// TwinCAT 3 PLC project JOGAN
// ProgramVersion: 3.1.4020.4
// libraries:
//   Tc2_Standard, * (Beckhoff Automation GmbH)
//   Tc2_System, * (Beckhoff Automation GmbH)
//   Tc3_Module, * (Beckhoff Automation GmbH)
// project tree:
//   DUTs/ T_MACHINE_POSITION.TcDUT, T_CURRENT_TRANSACTION.TcDUT, T_JIG_SOCKET.TcDUT
//   GVLs/ FLAG_VAR.TcGVL, INDEXING_1_VAR.TcGVL, INDEXING_2_VAR.TcGVL, INPUT_G6_VAR.TcGVL, INPUT_VAR.TcGVL, LOADER_RS4_VAR.TcGVL, LOADER_VAR.TcGVL, POWER_CONTROL.TcGVL, SORTER_RS4_VAR.TcGVL, SORTER_VAR.TcGVL, TESTER_C8_VAR.TcGVL
//   / PlcTask.TcTTO (not stored)
//   POUs/ EXECUTE_FUNCTION.TcPOU (not stored), MAIN.TcPOU, STQWE.TcPOU
//   POUs/FUKUDA/ FUKUDA_MOVE.TcPOU, FUKUDA_MOVE_1.TcPOU, INPUT_PROG.TcPOU, LOAD_FUKUDA.TcPOU, LOAD_FUKUDA_1.TcPOU, RETURN_FUKUDA.TcPOU, RETURN_FUKUDA_1.TcPOU (not stored)
//   POUs/LASER/ LASER_MOVE.TcPOU, LASER_PROG.TcPOU, LOAD_LASER.TcPOU, LOAD_NG.TcPOU, RETURN_LASER.TcPOU, RETURN_NG.TcPOU
//   POUs/LOADER/ INDEXING.TcPOU, INDEX_1.TcPOU, INDEXING_2.TcPOU, STRAIGHTENING_PROG_1.TcPOU, STR.TcPOU (not stored)
//   POUs/ROBOT/ INPUT_G6.TcPOU, TESTER_C8.TcPOU, LOADER_RS4.TcPOU, SORTER_RS4.TcPOU
// real-time tasks:
//   TASK PlcTask: cycle T#10ms, priority 20, ADS port 350
// I/O:
//   DEVICE Device 5 (EtherCAT), AmsNetId 172.18.128.227.6.1
//     Term 1 (EK1100) [EK1100 EtherCAT Coupler (2A E-Bus)]
//       Term 2 (EL1808) [EL1808 8Ch. Dig. Input 24V, 3ms]
//       Term 3 (EL1808) [EL1808 8Ch. Dig. Input 24V, 3ms]
//       Term 4 (EL1808) [EL1808 8Ch. Dig. Input 24V, 3ms]
//       Term 5 (EL1808) [EL1808 8Ch. Dig. Input 24V, 3ms]
//       Term 6 (EL2808) [EL2808 8Ch. Dig. Output 24V, 0.5A]
//       Term 7 (EL2808) [EL2808 8Ch. Dig. Output 24V, 0.5A]
//       Term 8 (EL2808) [EL2808 8Ch. Dig. Output 24V, 0.5A]
//       Term 9 (EL2808) [EL2808 8Ch. Dig. Output 24V, 0.5A]
//       Term 10 (EL2808) [EL2808 8Ch. Dig. Output 24V, 0.5A]
//       Term 11 (EL3058) [EL3058 8Ch. Ana. Input 4-20mA]
//       Term 12 (EL1904) [EL1904, 4 Ch. Safety Input 24V, TwinSAFE]
//         modules: Module 1 (FSOES)
//       Term 13 (EL1904) [EL1904, 4 Ch. Safety Input 24V, TwinSAFE]
//         modules: Module 1 (FSOES)
//       Term 14 (EL6731) [EL6731 PROFIBUS DP Master]
//       Term 15 (EK1110) [EK1110 EtherCAT extension]
//     Term 16 (EK1100) [EK1100 EtherCAT Coupler (2A E-Bus)]
//       Term 17 (EL1808) [EL1808 8Ch. Dig. Input 24V, 3ms]
//       Term 18 (EL1808) [EL1808 8Ch. Dig. Input 24V, 3ms]
//       Term 19 (EL1808) [EL1808 8Ch. Dig. Input 24V, 3ms]
//       Term 20 (EL1808) [EL1808 8Ch. Dig. Input 24V, 3ms]
//       Term 21 (EL1808) [EL1808 8Ch. Dig. Input 24V, 3ms]
//       Term 22 (EL1808) [EL1808 8K. Dig. Eingang 24V, 3ms]
//       Term 23 (EL2808) [EL2808 8Ch. Dig. Output 24V, 0.5A]
//       Term 24 (EL2808) [EL2808 8Ch. Dig. Output 24V, 0.5A]
//       Term 25 (EL2808) [EL2808 8Ch. Dig. Output 24V, 0.5A]
//       Term 26 (EL2808) [EL2808 8Ch. Dig. Output 24V, 0.5A]
//       Term 27 (EL2808) [EL2808 8Ch. Dig. Output 24V, 0.5A]
//       Term 28 (EL2808) [EL2808 8Ch. Dig. Output 24V, 0.5A]
//       Term 29 (EL2808) [EL2808 8Ch. Dig. Output 24V, 0.5A]
//       Term 30 (EL2808) [EL2808 8Ch. Dig. Output 24V, 0.5A]
//       Term 31 (EL6731) [EL6731 PROFIBUS DP Master]
//       Term 32 (EK1110) [EK1110 EtherCAT extension]
//     Box 33 (EP2809-0021)RS4-2 [EP2809-0021 16 Ch. Dig. Output 24V, 0,5A, M8]
//     Box 34 (EP1809-0021)RS4-2 [EP1809-0021 16 Ch. Dig. Input 24V, 3ms, M8]
//     Box 35 (EP2809-0021)RS4-1 [EP2809-0021 16 Ch. Dig. Output 24V, 0,5A, M8]
//     Box 36 (EP2809-0021)RS4-1 [EP1809-0021 16 Ch. Dig. Input 24V, 3ms, M8]
//     Box 37 (EP1809-0021)G6 [EP1809-0021 16 Ch. Dig. Input 24V, 3ms, M8]
//     Box 38 (EP2809-0021) G6 [EP2809-0021 16 Ch. Dig. Output 24V, 0,5A, M8]
//     Box 39 (EPSON RC700 EtherCAT Slave)G6 [EPSON RC700 EtherCAT Slave]
//     Box 40 (EPSON RC700 EtherCAT Slave)RS4-1 [EPSON RC700 EtherCAT Slave]
//     Box 40 (EPSON RC700 EtherCAT Slave)C8 [EPSON RC700 EtherCAT Slave]
//     Box 42 (EPSON RC700 EtherCAT Slave)RS4-2 [EPSON RC700 EtherCAT Slave]
//     Box 47 (EP2339-0021) [EP2339-0021 16 Ch. Dig. Input/Output 24V, 0,5A, M8]
//     Box 88 (EP2339-0021) [EP2339-0021 16 Ch. Dig. Input/Output 24V, 0,5A, M8]
//   DEVICE Device 1 (EL6731), AmsNetId 172.18.128.227.2.1
//     Box 43 (LEC-GPR1) // Vendor: SMC Corporation Revision: V1.0
//     Box 44 (AX9000T) INDEXING 1 // Vendor: CKD Corporation Revision: Version 1.000
//      // Vendor: CKD Corporation Revision: Version 1.000
//   DEVICE Device 2 (EL6731), AmsNetId 172.18.128.227.3.1
//     Box 46 (LEC-GPR1) // Vendor: SMC Corporation Revision: V1.0
// variable links:
//   JOGAN/JOGAN Instance <-> Device 1 (EL6731)/
//     PlcTask Inputs/INDEXING_2_VAR.DataByteInput2 <-> Module 1 (8 Bytes Out,8 Bytes In)/Inputs/8 Bytes Out,8 Bytes In_0_0
//     PlcTask Outputs/INDEXING_2_VAR.DataByteOutput2 <-> Module 1 (8 Bytes Out,8 Bytes In)/Outputs/8 Bytes Out,8 Bytes In_1_0
//   JOGAN/JOGAN Instance <-> Device 1 (EL6731)/Box 43 (LEC-GPR1)
//     PlcTask Inputs/INPUT_VAR.DataWordInput1 <-> Module 1 (Input 16 words)/Inputs/Input 16 words_0_0
//     PlcTask Inputs/INPUT_VAR.DataWordInput2 <-> Module 2 (Input 16 words)/Inputs/Input 16 words_0_0
//     PlcTask Inputs/INPUT_VAR.DataWordInput3 <-> Module 3 (Input 16 words)/Inputs/Input 16 words_0_0
//     PlcTask Outputs/INPUT_VAR.DataWordOutput1 <-> Module 5 (Output 16 words)/Outputs/Output 16 words_1_0
//     PlcTask Outputs/INPUT_VAR.DataWordOutput2 <-> Module 6 (Output 16 words)/Outputs/Output 16 words_1_0
//     PlcTask Outputs/INPUT_VAR.DataWordOutput3 <-> Module 7 (Output 16 words)/Outputs/Output 16 words_1_0
//     PlcTask Outputs/INPUT_VAR.DataWordOutput4 <-> Module 8 (Output 9 words)/Outputs/Output 9 words_1_0
//   JOGAN/JOGAN Instance <-> Device 1 (EL6731)/Box 44 (AX9000T) INDEXING 1
//     PlcTask Inputs/INDEXING_1_VAR.DataByteInput <-> Module 2 (8 Bytes Out,8 Bytes In)/Inputs/8 Bytes Out,8 Bytes In_0_0
//     PlcTask Outputs/INDEXING_1_VAR.DataByteOutput <-> Module 2 (8 Bytes Out,8 Bytes In)/Outputs/8 Bytes Out,8 Bytes In_1_0
//   JOGAN/JOGAN Instance <-> Device 2 (EL6731)/Box 46 (LEC-GPR1)
//     PlcTask Inputs/SORTER_VAR.DataWordInput1 <-> Module 1 (Input 16 words)/Inputs/Input 16 words_0_0
//     PlcTask Inputs/SORTER_VAR.DataWordInput2 <-> Module 2 (Input 16 words)/Inputs/Input 16 words_0_0
//     PlcTask Inputs/SORTER_VAR.DataWordInput3 <-> Module 3 (Input 16 words)/Inputs/Input 16 words_0_0
//     PlcTask Inputs/SORTER_VAR.DataWordInput4 <-> Module 4 (Input 9 words)/Inputs/Input 9 words_0_0
//     PlcTask Outputs/SORTER_VAR.DataWordOutput1 <-> Module 5 (Output 16 words)/Outputs/Output 16 words_1_0
//     PlcTask Outputs/SORTER_VAR.DataWordOutput2 <-> Module 6 (Output 16 words)/Outputs/Output 16 words_1_0
//     PlcTask Outputs/SORTER_VAR.DataWordOutput3 <-> Module 7 (Output 16 words)/Outputs/Output 16 words_1_0
//     PlcTask Outputs/SORTER_VAR.DataWordOutput4 <-> Module 8 (Output 9 words)/Outputs/Output 9 words_1_0
//   JOGAN/JOGAN Instance <-> Device 5 (EtherCAT)/Box 33 (EP2809-0021)RS4-2
//     PlcTask Outputs/SORTER_RS4_VAR.O_SORTER_RS4_GRIPPER_CLOSE_{1..4} <-> Channel {1..7 step 2}/Output  (4 links)
//     PlcTask Outputs/SORTER_RS4_VAR.O_SORTER_RS4_GRIPPER_EXT_DOWN_{1..4} <-> Channel {9..15 step 2}/Output  (4 links)
//     PlcTask Outputs/SORTER_RS4_VAR.O_SORTER_RS4_GRIPPER_EXT_UP_{1..4} <-> Channel {10..16 step 2}/Output  (4 links)
//     PlcTask Outputs/SORTER_RS4_VAR.O_SORTER_RS4_GRIPPER_OPEN_{1..4} <-> Channel {2..8 step 2}/Output  (4 links)
//   JOGAN/JOGAN Instance <-> Device 5 (EtherCAT)/Box 34 (EP1809-0021)RS4-2
//     PlcTask Inputs/SORTER_RS4_VAR.I_SORTER_RS4_GRIPPER_CLOSE_{1..4} <-> Channel {2..8 step 2}/Input  (4 links)
//     PlcTask Inputs/SORTER_RS4_VAR.I_SORTER_RS4_GRIPPER_EXT_DOWN_{1..4} <-> Channel {10..16 step 2}/Input  (4 links)
//     PlcTask Inputs/SORTER_RS4_VAR.I_SORTER_RS4_GRIPPER_EXT_UP_{1..4} <-> Channel {9..15 step 2}/Input  (4 links)
//     PlcTask Inputs/SORTER_RS4_VAR.I_SORTER_RS4_GRIPPER_OPEN_{1..4} <-> Channel {1..7 step 2}/Input  (4 links)
//   JOGAN/JOGAN Instance <-> Device 5 (EtherCAT)/Box 35 (EP2809-0021)RS4-1
//     PlcTask Outputs/LOADER_RS4_VAR.O_LOADER_RS4_GRIPPER_CLOSE_{1..4} <-> Channel {1..7 step 2}/Output  (4 links)
//     PlcTask Outputs/LOADER_RS4_VAR.O_LOADER_RS4_GRIPPER_EXT_DOWN_{1..4} <-> Channel {9..15 step 2}/Output  (4 links)
//     PlcTask Outputs/LOADER_RS4_VAR.O_LOADER_RS4_GRIPPER_EXT_UP_{1..4} <-> Channel {10..16 step 2}/Output  (4 links)
//     PlcTask Outputs/LOADER_RS4_VAR.O_LOADER_RS4_GRIPPER_OPEN_{1..4} <-> Channel {2..8 step 2}/Output  (4 links)
//   JOGAN/JOGAN Instance <-> Device 5 (EtherCAT)/Box 36 (EP2809-0021)RS4-1
//     PlcTask Inputs/LOADER_RS4_VAR.I_LOADER_RS4_GRIPPER_CLOSE_{1..4} <-> Channel {10..16 step 2}/Input  (4 links)
//     PlcTask Inputs/LOADER_RS4_VAR.I_LOADER_RS4_GRIPPER_EXT_DOWN_{1..4} <-> Channel {2..8 step 2}/Input  (4 links)
//     PlcTask Inputs/LOADER_RS4_VAR.I_LOADER_RS4_GRIPPER_EXT_UP_{1..4} <-> Channel {1..7 step 2}/Input  (4 links)
//     PlcTask Inputs/LOADER_RS4_VAR.I_LOADER_RS4_GRIPPER_OPEN_{1..4} <-> Channel {9..15 step 2}/Input  (4 links)
//   JOGAN/JOGAN Instance <-> Device 5 (EtherCAT)/Box 37 (EP1809-0021)G6
//     PlcTask Inputs/INPUT_G6_VAR.I_G6_GRIPPER_CLOSE_{1..4} <-> Channel {10..16 step 2}/Input  (4 links)
//     PlcTask Inputs/INPUT_G6_VAR.I_G6_GRIPPER_EXT_DOWN_{1..4} <-> Channel {2..8 step 2}/Input  (4 links)
//     PlcTask Inputs/INPUT_G6_VAR.I_G6_GRIPPER_EXT_UP_{1..4} <-> Channel {1..7 step 2}/Input  (4 links)
//     PlcTask Inputs/INPUT_G6_VAR.I_G6_GRIPPER_OPEN_{1..4} <-> Channel {9..15 step 2}/Input  (4 links)
//   JOGAN/JOGAN Instance <-> Device 5 (EtherCAT)/Box 38 (EP2809-0021) G6
//     PlcTask Outputs/INPUT_G6_VAR.O_G6_GRIPPER_CLOSE_{1..4} <-> Channel {1..7 step 2}/Output  (4 links)
//     PlcTask Outputs/INPUT_G6_VAR.O_G6_GRIPPER_EXT_DOWN_{1..4} <-> Channel {9..15 step 2}/Output  (4 links)
//     PlcTask Outputs/INPUT_G6_VAR.O_G6_GRIPPER_EXT_UP_{1..4} <-> Channel {10..16 step 2}/Output  (4 links)
//     PlcTask Outputs/INPUT_G6_VAR.O_G6_GRIPPER_OPEN_{1..4} <-> Channel {2..8 step 2}/Output  (4 links)
//   JOGAN/JOGAN Instance <-> Device 5 (EtherCAT)/Box 39 (EPSON RC700 EtherCAT Slave)G6
//     PlcTask Inputs/INPUT_G6_VAR.COUNTER_FUKUDA_A <-> TxPDO/Input byte 0006
//     PlcTask Inputs/INPUT_G6_VAR.COUNTER_FUKUDA_B <-> TxPDO/Input byte 0007
//     PlcTask Inputs/INPUT_G6_VAR.G6_ERROR1 <-> TxPDO/Input byte 0002
//     PlcTask Inputs/INPUT_G6_VAR.G6_ERROR2 <-> TxPDO/Input byte 0003
//     PlcTask Inputs/INPUT_G6_VAR.G6_INPUT <-> TxPDO/Input byte 0000
//     PlcTask Inputs/INPUT_G6_VAR.G6_INPUT_1 <-> TxPDO/Input byte 0001
//     PlcTask Inputs/INPUT_G6_VAR.G6_INPUT_2 <-> TxPDO/Input byte 0004
//     PlcTask Inputs/INPUT_G6_VAR.G6_INPUT_3 <-> TxPDO/Input byte 0005
//     PlcTask Outputs/INPUT_G6_VAR.G6_OUTPUT <-> RxPDO/Output byte 0000
//     PlcTask Outputs/INPUT_G6_VAR.G6_OUTPUT_1 <-> RxPDO/Output byte 0001
//     PlcTask Outputs/INPUT_G6_VAR.G6_OUTPUT_2 <-> RxPDO/Output byte 0002
//     PlcTask Outputs/INPUT_G6_VAR.START_POSITION <-> RxPDO/Output byte 0010
//   JOGAN/JOGAN Instance <-> Device 5 (EtherCAT)/Box 40 (EPSON RC700 EtherCAT Slave)C8
//     PlcTask Inputs/TESTER_C8_VAR.C8_ERROR_1 <-> TxPDO/Input byte 0002
//     PlcTask Inputs/TESTER_C8_VAR.C8_ERROR_2 <-> TxPDO/Input byte 0003
//     PlcTask Inputs/TESTER_C8_VAR.C8_INPUT_1 <-> TxPDO/Input byte 0004
//     PlcTask Inputs/TESTER_C8_VAR.C8_STATE_1 <-> TxPDO/Input byte 0000
//     PlcTask Inputs/TESTER_C8_VAR.C8_STATE_2 <-> TxPDO/Input byte 0001
//     PlcTask Outputs/TESTER_C8_VAR.C8_CONTROL_1 <-> RxPDO/Output byte 0000
//     PlcTask Outputs/TESTER_C8_VAR.C8_CONTROL_2 <-> RxPDO/Output byte 0001
//     PlcTask Outputs/TESTER_C8_VAR.C8_CONTROL_3 <-> RxPDO/Output byte 0002
//     PlcTask Outputs/TESTER_C8_VAR.C8_INDEX_POSITION <-> RxPDO/Output byte 0003
//     PlcTask Outputs/TESTER_C8_VAR.C8_MOVEMENT_DESTINATION <-> RxPDO/Output byte 0005
//     PlcTask Outputs/TESTER_C8_VAR.C8_MOVEMENT_SOURCE <-> RxPDO/Output byte 0004
//   JOGAN/JOGAN Instance <-> Device 5 (EtherCAT)/Box 40 (EPSON RC700 EtherCAT Slave)RS4-1
//     PlcTask Inputs/LOADER_RS4_VAR.LOADER_RS4_INPUT <-> TxPDO/Input byte 0000
//     PlcTask Inputs/LOADER_RS4_VAR.LOADER_RS4_INPUT_1 <-> TxPDO/Input byte 0001
//     PlcTask Inputs/LOADER_RS4_VAR.LOADER_RS4_INPUT_2 <-> TxPDO/Input byte 0004
//     PlcTask Inputs/LOADER_RS4_VAR.LOADER_RS4_INPUT_3 <-> TxPDO/Input byte 0005
//     PlcTask Outputs/LOADER_RS4_VAR.CARRIER_INDEX <-> RxPDO/Output byte 0006
//     PlcTask Outputs/LOADER_RS4_VAR.GRIPPER_SENSOR <-> RxPDO/Output byte 0008
//     PlcTask Outputs/LOADER_RS4_VAR.LOADER_RS4_OUTPUT <-> RxPDO/Output byte 0000
//     PlcTask Outputs/LOADER_RS4_VAR.LOADER_RS4_OUTPUT_1 <-> RxPDO/Output byte 0001
//     PlcTask Outputs/LOADER_RS4_VAR.LOADER_RS4_OUTPUT_2 <-> RxPDO/Output byte 0007
//     PlcTask Outputs/LOADER_RS4_VAR.POSITION_TOOL_1 <-> RxPDO/Output byte 0002
//     PlcTask Outputs/LOADER_RS4_VAR.POSITION_TOOL_2 <-> RxPDO/Output byte 0003
//     PlcTask Outputs/LOADER_RS4_VAR.POSITION_TOOL_3 <-> RxPDO/Output byte 0004
//     PlcTask Outputs/LOADER_RS4_VAR.POSITION_TOOL_4 <-> RxPDO/Output byte 0005
//   JOGAN/JOGAN Instance <-> Device 5 (EtherCAT)/Box 42 (EPSON RC700 EtherCAT Slave)RS4-2
//     PlcTask Inputs/SORTER_RS4_VAR.SORTER_RS4_INPUT <-> TxPDO/Input byte 0000
//     PlcTask Inputs/SORTER_RS4_VAR.SORTER_RS4_INPUT_1 <-> TxPDO/Input byte 0001
//     PlcTask Inputs/SORTER_RS4_VAR.SORTER_RS4_INPUT_2 <-> TxPDO/Input byte 0004
//     PlcTask Inputs/SORTER_RS4_VAR.SORTER_RS4_INPUT_3 <-> TxPDO/<empty>
//     PlcTask Outputs/SORTER_RS4_VAR.SORTER_RS4_OUTPUT <-> RxPDO/Output byte 0000
//     PlcTask Outputs/SORTER_RS4_VAR.SORTER_RS4_OUTPUT_1 <-> RxPDO/Output byte 0001
//     PlcTask Outputs/SORTER_RS4_VAR.SORTER_RS4_POS_PLACING_1 <-> RxPDO/Output byte 0006
//     PlcTask Outputs/SORTER_RS4_VAR.SORTER_RS4_POS_PLACING_2 <-> RxPDO/Output byte 0007
//     PlcTask Outputs/SORTER_RS4_VAR.SORTER_RS4_POS_PLACING_3 <-> RxPDO/Output byte 0008
//     PlcTask Outputs/SORTER_RS4_VAR.SORTER_RS4_POS_PLACING_4 <-> RxPDO/Output byte 0009
//     PlcTask Outputs/SORTER_RS4_VAR.SORTER_RS4_POS_TAKEUP_1 <-> RxPDO/Output byte 0002
//     PlcTask Outputs/SORTER_RS4_VAR.SORTER_RS4_POS_TAKEUP_2 <-> RxPDO/Output byte 0003
//     PlcTask Outputs/SORTER_RS4_VAR.SORTER_RS4_POS_TAKEUP_3 <-> RxPDO/Output byte 0004
//     PlcTask Outputs/SORTER_RS4_VAR.SORTER_RS4_POS_TAKEUP_4 <-> RxPDO/Output byte 0005
//   JOGAN/JOGAN Instance <-> Device 5 (EtherCAT)/Box 47 (EP2339-0021)
//     PlcTask Inputs/LOADER_VAR.I_C8_GRIPPER_OFF <-> Channel 3/Input
//     PlcTask Inputs/LOADER_VAR.I_C8_GRIPPER_ON <-> Channel 4/Input
//     PlcTask Outputs/TESTER_C8_VAR.O_C8_GRIPPER_CLOSE <-> Channel 17/Output
//     PlcTask Outputs/TESTER_C8_VAR.O_C8_GRIPPER_OPEN <-> Channel 18/Output
//   JOGAN/JOGAN Instance <-> Device 5 (EtherCAT)/Box 88 (EP2339-0021)
//     PlcTask Inputs/LOADER_VAR.I_TESTER_JIG_PRESENCE_11 <-> Channel 10/Input
//   JOGAN/JOGAN Instance <-> Device 5 (EtherCAT)/Term 1 (EK1100)/Term 10 (EL2808)
//     PlcTask Outputs/INPUT_VAR.O_RESET_CARTESSIAN <-> Channel 3/Output
//     PlcTask Outputs/INPUT_VAR.O_STOPPER_TRANSFER_A <-> Channel 1/Output
//     PlcTask Outputs/INPUT_VAR.O_STOPPER_TRANSFER_B <-> Channel 2/Output
//   JOGAN/JOGAN Instance <-> Device 5 (EtherCAT)/Term 1 (EK1100)/Term 2 (EL1808)
//     PlcTask Inputs/INPUT_VAR.I_FUKUDA_TRANSFER_AT_BACK_A <-> Channel 3/Input
//     PlcTask Inputs/INPUT_VAR.I_FUKUDA_TRANSFER_AT_BACK_B <-> Channel 1/Input
//     PlcTask Inputs/INPUT_VAR.I_FUKUDA_TRANSFER_AT_FRONT_A <-> Channel 4/Input
//     PlcTask Inputs/INPUT_VAR.I_FUKUDA_TRANSFER_AT_FRONT_B <-> Channel 2/Input
//     PlcTask Inputs/INPUT_VAR.I_LOTBOX_DETECT_{1..4} <-> Channel {5..8}/Input  (4 links)
//   JOGAN/JOGAN Instance <-> Device 5 (EtherCAT)/Term 1 (EK1100)/Term 3 (EL1808)
//     PlcTask Inputs/INDEXING_1_VAR.I_INDEXING_1_GRIPPER_CLOSE_{1..4} <-> Channel {1..7 step 2}/Input  (4 links)
//     PlcTask Inputs/INDEXING_1_VAR.I_INDEXING_1_GRIPPER_OPEN_{1..4} <-> Channel {2..8 step 2}/Input  (4 links)
//   JOGAN/JOGAN Instance <-> Device 5 (EtherCAT)/Term 1 (EK1100)/Term 4 (EL1808)
//     PlcTask Inputs/INDEXING_1_VAR.I_INDEXING_1_GRIPPER_EXT_DOWN <-> Channel 2/Input
//     PlcTask Inputs/INDEXING_1_VAR.I_INDEXING_1_GRIPPER_EXT_UP <-> Channel 1/Input
//     PlcTask Inputs/INPUT_VAR.I_LOTBOX_CLAMP_OFF_1 <-> Channel 6/Input
//     PlcTask Inputs/INPUT_VAR.I_LOTBOX_CLAMP_OFF_2 <-> Channel 8/Input
//     PlcTask Inputs/INPUT_VAR.I_LOTBOX_CLAMP_ON_1 <-> Channel 5/Input
//     PlcTask Inputs/INPUT_VAR.I_LOTBOX_CLAMP_ON_2 <-> Channel 7/Input
//   JOGAN/JOGAN Instance <-> Device 5 (EtherCAT)/Term 1 (EK1100)/Term 5 (EL1808)
//     PlcTask Inputs/INDEXING_1_VAR.I_PRESS_STOPPER_DOWN <-> Channel 7/Input
//     PlcTask Inputs/INDEXING_1_VAR.I_PRESS_STOPPER_UP <-> Channel 8/Input
//     PlcTask Inputs/INPUT_VAR.I_LOTBOX_CLAMP_OFF_3 <-> Channel 2/Input
//     PlcTask Inputs/INPUT_VAR.I_LOTBOX_CLAMP_OFF_4 <-> Channel 4/Input
//     PlcTask Inputs/INPUT_VAR.I_LOTBOX_CLAMP_ON_3 <-> Channel 1/Input
//     PlcTask Inputs/INPUT_VAR.I_LOTBOX_CLAMP_ON_4 <-> Channel 3/Input
//     PlcTask Inputs/INPUT_VAR.I_VACUUM_OFF <-> Channel 6/Input
//     PlcTask Inputs/INPUT_VAR.I_VACUUM_ON <-> Channel 5/Input
//   JOGAN/JOGAN Instance <-> Device 5 (EtherCAT)/Term 1 (EK1100)/Term 6 (EL2808)
//     PlcTask Outputs/INPUT_VAR.O_TOWER_LAMP_BUZZER <-> Channel 8/Output
//     PlcTask Outputs/INPUT_VAR.O_TOWER_LAMP_GREEN <-> Channel 7/Output
//     PlcTask Outputs/INPUT_VAR.O_TOWER_LAMP_RED <-> Channel 5/Output
//     PlcTask Outputs/INPUT_VAR.O_TOWER_LAMP_YELLOW <-> Channel 6/Output
//     PlcTask Outputs/INPUT_VAR.O_VACUUM_OFF <-> Channel 2/Output
//     PlcTask Outputs/INPUT_VAR.O_VACUUM_ON <-> Channel 1/Output
//   JOGAN/JOGAN Instance <-> Device 5 (EtherCAT)/Term 1 (EK1100)/Term 7 (EL2808)
//     PlcTask Outputs/INDEXING_1_VAR.O_INDEXING_1_GRIPPER_CLOSE_{1..4} <-> Channel {1..7 step 2}/Output  (4 links)
//     PlcTask Outputs/INDEXING_1_VAR.O_INDEXING_1_GRIPPER_OPEN_{1..4} <-> Channel {2..8 step 2}/Output  (4 links)
//   JOGAN/JOGAN Instance <-> Device 5 (EtherCAT)/Term 1 (EK1100)/Term 8 (EL2808)
//     PlcTask Outputs/INDEXING_1_VAR.O_INDEXING_1_GRIPPER_EXT_DOWN <-> Channel 2/Output
//     PlcTask Outputs/INDEXING_1_VAR.O_INDEXING_1_GRIPPER_EXT_UP <-> Channel 1/Output
//     PlcTask Outputs/INDEXING_1_VAR.O_PRESS_STOPPER_DOWN <-> Channel 7/Output
//     PlcTask Outputs/INDEXING_1_VAR.O_PRESS_STOPPER_UP <-> Channel 8/Output
//     PlcTask Outputs/INPUT_VAR.O_LOT_BOX_INDICATOR_{1..4} <-> Channel {3..6}/Output  (4 links)
//   JOGAN/JOGAN Instance <-> Device 5 (EtherCAT)/Term 1 (EK1100)/Term 9 (EL2808)
//     PlcTask Outputs/INPUT_VAR.O_LOTBOX_CLAMP_OFF_{1..4} <-> Channel {7..1 step -2}/Output  (4 links)
//     PlcTask Outputs/INPUT_VAR.O_LOTBOX_CLAMP_ON_{1..4} <-> Channel {8..2 step -2}/Output  (4 links)
//   JOGAN/JOGAN Instance <-> Device 5 (EtherCAT)/Term 16 (EK1100)/Term 18 (EL1808)
//     PlcTask Inputs/LOADER_VAR.I_CARRIER_DETECT_{1..4} <-> Channel {1..4}/Input  (4 links)
//     PlcTask Inputs/SORTER_VAR.I_NG_BOX_DETECT_{1..4} <-> Channel {5..8}/Input  (4 links)
//   JOGAN/JOGAN Instance <-> Device 5 (EtherCAT)/Term 16 (EK1100)/Term 19 (EL1808)
//     PlcTask Inputs/SORTER_VAR.I_CARTESSIAN_GRIPPER_OFF <-> Channel 2/Input
//     PlcTask Inputs/SORTER_VAR.I_CARTESSIAN_GRIPPER_ON <-> Channel 1/Input
//     PlcTask Inputs/SORTER_VAR.I_LASER_TRANSFER_AT_BACK_A <-> Channel 7/Input
//     PlcTask Inputs/SORTER_VAR.I_LASER_TRANSFER_AT_FRONT_A <-> Channel 6/Input
//     PlcTask Inputs/SORTER_VAR.I_LASER_TRANSFER_AT_FRONT_B <-> Channel 8/Input
//     PlcTask Inputs/SORTER_VAR.I_NG_BUFFER_OFF <-> Channel 3/Input
//     PlcTask Inputs/SORTER_VAR.I_NG_BUFFER_ON <-> Channel 4/Input
//   JOGAN/JOGAN Instance <-> Device 5 (EtherCAT)/Term 16 (EK1100)/Term 20 (EL1808)
//     PlcTask Inputs/SORTER_VAR.I_LASER_TRANSFER_AT_BACK_B <-> Channel 1/Input
//     PlcTask Inputs/SORTER_VAR.I_NG_TRANSFER_AT_BACK <-> Channel 3/Input
//     PlcTask Inputs/SORTER_VAR.I_NG_TRANSFER_AT_FRONT <-> Channel 2/Input
//   JOGAN/JOGAN Instance <-> Device 5 (EtherCAT)/Term 16 (EK1100)/Term 21 (EL1808)
//     PlcTask Inputs/SORTER_VAR.I_LOTBOX_DETECT_{1..4} <-> Channel {4..7}/Input  (4 links)
//   JOGAN/JOGAN Instance <-> Device 5 (EtherCAT)/Term 16 (EK1100)/Term 23 (EL2808)
//     PlcTask Outputs/SORTER_VAR.O_LOTBOX_CLAMP_OFF_{1..4} <-> Channel {2..8 step 2}/Output  (4 links)
//     PlcTask Outputs/SORTER_VAR.O_LOTBOX_CLAMP_ON_{1..4} <-> Channel {1..7 step 2}/Output  (4 links)
//   JOGAN/JOGAN Instance <-> Device 5 (EtherCAT)/Term 16 (EK1100)/Term 24 (EL2808)
//     PlcTask Outputs/SORTER_VAR.O_CARTESSIAN_GRIPPER_OFF <-> Channel 4/Output
//     PlcTask Outputs/SORTER_VAR.O_CARTESSIAN_GRIPPER_ON <-> Channel 3/Output
//   JOGAN/JOGAN Instance <-> Device 5 (EtherCAT)/Term 16 (EK1100)/Term 25 (EL2808)
//     PlcTask Outputs/SORTER_VAR.O_LOT_BOX_INDICATOR_1 <-> Channel 6/Output
//     PlcTask Outputs/SORTER_VAR.O_LOT_BOX_INDICATOR_2 <-> Channel 7/Output
//     PlcTask Outputs/SORTER_VAR.O_LOT_BOX_INDICATOR_3 <-> Channel 8/Output
//     PlcTask Outputs/SORTER_VAR.O_TOWER_LAMP_BUZZER <-> Channel 4/Output
//     PlcTask Outputs/SORTER_VAR.O_TOWER_LAMP_GREEN <-> Channel 1/Output
//     PlcTask Outputs/SORTER_VAR.O_TOWER_LAMP_RED <-> Channel 2/Output
//     PlcTask Outputs/SORTER_VAR.O_TOWER_LAMP_YELLOW <-> Channel 3/Output
//   JOGAN/JOGAN Instance <-> Device 5 (EtherCAT)/Term 16 (EK1100)/Term 26 (EL2808)
//     PlcTask Outputs/SORTER_VAR.O_LOT_BOX_INDICATOR_4 <-> Channel 1/Output
//     PlcTask Outputs/SORTER_VAR.O_NG_BUFFER_OFF <-> Channel 4/Output
//     PlcTask Outputs/SORTER_VAR.O_NG_BUFFER_ON <-> Channel 3/Output
//     PlcTask Outputs/SORTER_VAR.O_NG_DATA_OUTPUT{1..4} <-> Channel {5..8}/Output  (4 links)
//   JOGAN/JOGAN Instance <-> Device 5 (EtherCAT)/Term 16 (EK1100)/Term 29 (EL2808)
//     PlcTask Outputs/POWER_CONTROL.O_PWR_CTRL_INDEXING_1 <-> Channel 7/Output
//     PlcTask Outputs/POWER_CONTROL.O_PWR_CTRL_INDEXING_2 <-> Channel 8/Output
//     PlcTask Outputs/POWER_CONTROL.O_PWR_CTRL_ROBOT_C8 <-> Channel 6/POWER_CONTROL.O_PWR_CTRL_ROBOT_C8
//     PlcTask Outputs/POWER_CONTROL.O_PWR_CTRL_ROBOT_G6 <-> Channel 3/Output
//     PlcTask Outputs/POWER_CONTROL.O_PWR_CTRL_ROBOT_RS4_1 <-> Channel 4/Output
//     PlcTask Outputs/POWER_CONTROL.O_PWR_CTRL_ROBOT_RS4_2 <-> Channel 5/Output
//   JOGAN/JOGAN Instance <-> Device 5 (EtherCAT)/Term 16 (EK1100)/Term 30 (EL2808)
//     PlcTask Outputs/SORTER_VAR.O_NG_BOX_INDICATOR_1 <-> Channel 3/<empty>
//     PlcTask Outputs/SORTER_VAR.O_NG_BOX_INDICATOR_2 <-> Channel 4/Output
//     PlcTask Outputs/SORTER_VAR.O_NG_BOX_INDICATOR_3 <-> Channel 5/Output
//     PlcTask Outputs/SORTER_VAR.O_NG_BOX_INDICATOR_4 <-> Channel 6/Output
//     PlcTask Outputs/SORTER_VAR.O_RESET_CARTESSIAN <-> Channel 8/Output
//     PlcTask Outputs/SORTER_VAR.O_STOPPER_TRANSFER_A <-> Channel 1/Output
//     PlcTask Outputs/SORTER_VAR.O_STOPPER_TRANSFER_B <-> Channel 2/Output

// ---- DUTs/T_MACHINE_POSITION.TcDUT
TYPE T_MACHINE_POSITION :
STRUCT
	DESTINATION_COORDINATE:BYTE:=11;	
	SUB_DESTINATION_COORDINATE:BYTE:=0;	
	SOURCE_COORDINATE:BYTE:=0;
END_STRUCT
END_TYPE

// ---- DUTs/T_CURRENT_TRANSACTION.TcDUT
TYPE T_CURRENT_TRANSACTION :
STRUCT
	STATION_NUMBER_LOAD : BYTE :=1;
	STATION_NUMBER_RETURN : BYTE :=1;
    CURRENT_DEVICE_COUNT : BYTE :=0;
	QUANTITY_MAX : BYTE :=0;
	QUANTITY_LOTEND :BYTE :=0;
	JIG_INDEX_LOAD : BYTE :=1;
	JIG_INDEX_RETURN : BYTE :=1;
	JIG_INDEX_LOAD_NG : BYTE :=1;
	JIG_INDEX_RETURN_NG : BYTE :=1;
	TRANSPORT_INDEX : BYTE :=1;
	PO_NUMBER : STRING[255] := '';
END_STRUCT
END_TYPE

// ---- DUTs/T_JIG_SOCKET.TcDUT
TYPE T_JIG_SOCKET :
STRUCT
	STATION_NUMBER:BYTE:=0;
	CURRENT_DEVICE_COUNT : BYTE :=0;
	MAX_DEVICE_COUNT : BYTE :=0;
	AVAILABLE_SOCKET : ARRAY[0..4] OF BYTE;
	LASER_DESTINATION: ARRAY[0..4] OF BYTE;
	PO_NUMBER : STRING[255] := '';
	
END_STRUCT
END_TYPE

// ---- GVLs/FLAG_VAR.TcGVL
  {attribute 'qualified_only'}
VAR_GLOBAL
	ALLOW_EXECUTE_LOAD_FUKUDA : BOOL:=FALSE;
	ALLOW_EXECUTE_RETURN_FUKUDA:BOOL:=FALSE;

	
	ALLOW_EXECUTE_LOAD_LASER:BOOL:=FALSE;
	ALLOW_EXECUTE_RETURN_LASER:BOOL:=FALSE;
	
	ALLOW_EXECUTE_LOAD_NG : BOOL:=FALSE;
	ALLOW_EXECUTE_RETURN_NG:BOOL:=FALSE;
	ALLOW_EXECUTE_C8:BOOL:=FALSE;
	PAUSE_SYSTEM:BOOL:=FALSE;
END_VAR

// ---- GVLs/INDEXING_1_VAR.TcGVL
{attribute 'qualified_CLOSEly'}
VAR_GLOBAL
	
I_INDEXING_1_GRIPPER_CLOSE_1 AT %I* : BOOL;
I_INDEXING_1_GRIPPER_CLOSE_2 AT %I* : BOOL;
I_INDEXING_1_GRIPPER_CLOSE_3 AT %I* : BOOL;
I_INDEXING_1_GRIPPER_CLOSE_4 AT %I* : BOOL;
I_INDEXING_1_GRIPPER_OPEN_1 AT %I* : BOOL;
I_INDEXING_1_GRIPPER_OPEN_2 AT %I* : BOOL;
I_INDEXING_1_GRIPPER_OPEN_3 AT %I* : BOOL;
I_INDEXING_1_GRIPPER_OPEN_4 AT %I* : BOOL;
I_INDEXING_1_GRIPPER_EXT_UP AT %I* : BOOL;
I_INDEXING_1_GRIPPER_EXT_DOWN AT %I* : BOOL;

O_INDEXING_1_GRIPPER_EXT_UP AT %Q* : BOOL;
O_INDEXING_1_GRIPPER_EXT_DOWN AT %Q* : BOOL;
O_INDEXING_1_GRIPPER_CLOSE_1 AT %Q* : BOOL;
O_INDEXING_1_GRIPPER_CLOSE_2 AT %Q* : BOOL;
O_INDEXING_1_GRIPPER_CLOSE_3 AT %Q* : BOOL;
O_INDEXING_1_GRIPPER_CLOSE_4 AT %Q* : BOOL;
O_INDEXING_1_GRIPPER_OPEN_1 AT %Q* : BOOL;
O_INDEXING_1_GRIPPER_OPEN_2 AT %Q* : BOOL;
O_INDEXING_1_GRIPPER_OPEN_3 AT %Q* : BOOL;
O_INDEXING_1_GRIPPER_OPEN_4 AT %Q* : BOOL;

I_PRESS_STOPPER_DOWN AT %I* : BOOL;
I_PRESS_STOPPER_UP AT %I* : BOOL;

O_PRESS_STOPPER_DOWN AT %Q* : BOOL;
O_PRESS_STOPPER_UP AT %Q* : BOOL;

O_INDEXING_1_HOME   : BOOL;
O_ROTATION_START : BOOL;
O_ROTATION_STOP : BOOL;

I_INDEXING_1_READY_FOR_STRAIGHTEN: BOOL;
I_INDEXING_1_HOME : BOOL;
O_INDEXING_1_POWER_OFF AT %Q* : BOOL;

I_INDEXING_1_ROTATION_START: BOOL;
I_INDEXING_1_ROTATION_PROCESS: BOOL;
I_INDEXING_1_ROTATION_DONE: BOOL ;

I_ALL_GRIPPER_OPEN: BOOL;
NUMBER_OF_STRAIGHTEN: INT :=0;
INDEXING_1_CASE: INT ;
TOTALNUMBER_OF_STRAIGHTEN :INT :=1;
STRAIGHTEN_FINISH:BOOL;
READY_STRAIGTHEN: BOOL;

DataByteOutput AT%Q* : ARRAY[0..7] OF BYTE;
DataByteInput AT%I* : ARRAY[0..7] OF BYTE;
END_VAR

// ---- GVLs/INDEXING_2_VAR.TcGVL
{attribute 'qualified_CLOSEly'}
VAR_GLOBAL
	
I_INDEXING_22_GRIPPER_CLOSE_1 AT %I* : BOOL;
I_INDEXING_2_GRIPPER_CLOSE_2 AT %I* : BOOL;
I_INDEXING_2_GRIPPER_CLOSE_3 AT %I* : BOOL;
I_INDEXING_2_GRIPPER_CLOSE_4 AT %I* : BOOL;
I_INDEXING_2_GRIPPER_OPEN_1 AT %I* : BOOL;
I_INDEXING_2_GRIPPER_OPEN_2 AT %I* : BOOL;
I_INDEXING_2_GRIPPER_OPEN_3 AT %I* : BOOL;
I_INDEXING_2_GRIPPER_OPEN_4 AT %I* : BOOL;
I_INDEXING_2_GRIPPER_EXT_UP AT %I* : BOOL;
I_INDEXING_2_GRIPPER_EXT_DOWN AT %I* : BOOL;

O_INDEXING_2_GRIPPER_EXT_UP AT %Q* : BOOL;
O_INDEXING_2_GRIPPER_EXT_DOWN AT %Q* : BOOL;
O_INDEXING_2_GRIPPER_CLOSE_1 AT %Q* : BOOL;
O_INDEXING_2_GRIPPER_CLOSE_2 AT %Q* : BOOL;
O_INDEXING_2_GRIPPER_CLOSE_3 AT %Q* : BOOL;
O_INDEXING_2_GRIPPER_CLOSE_4 AT %Q* : BOOL;
O_INDEXING_2_GRIPPER_OPEN_1 AT %Q* : BOOL;
O_INDEXING_2_GRIPPER_OPEN_2 AT %Q* : BOOL;
O_INDEXING_2_GRIPPER_OPEN_3 AT %Q* : BOOL;
O_INDEXING_2_GRIPPER_OPEN_4 AT %Q* : BOOL;

I_PRESS_STOPPER_DOWN AT %I* : BOOL;
I_PRESS_STOPPER_UP AT %I* : BOOL;

O_PRESS_STOPPER_DOWN AT %Q* : BOOL;
O_PRESS_STOPPER_UP AT %Q* : BOOL;

O_INDEXING_HOME   : BOOL;
O_ROTATION_DONE : BOOL;
O_ROTATION_START : BOOL;
O_ROTATION_STOP : BOOL;

I_INDEXING_2_READY_FOR_STRAIGHTEN: BOOL;
I_INDEXING_2_HOME : BOOL;
O_INDEXING_2_POWER_OFF AT %Q* : BOOL;

I_INDEXING_2_ROTATION_DONE: BOOL :=TRUE;
I_ALL_GRIPPER_OPEN: BOOL;
NUMBER_OF_STRAIGHTEN: INT :=0;
INDEXING_2_CASE: INT ;
TOTALNUMBER_OF_STRAIGHTEN :INT :=1;
CARRIER_INDEX: BYTE;

DataByteOutput2 AT%Q* : ARRAY[0..7] OF BYTE;
DataByteInput2 AT%I* : ARRAY[0..7] OF BYTE;
END_VAR

// ---- GVLs/INPUT_G6_VAR.TcGVL
{attribute 'qualified_only'}
VAR_GLOBAL
G6_INPUT AT %IB00 :  	BYTE;
G6_INPUT_1 AT %IB01 : 	BYTE;
G6_INPUT_2 AT %IB02 : 	BYTE;
G6_INPUT_3 AT %IB03 :	BYTE;
COUNTER_FUKUDA_A AT %IB06 :	BYTE;
COUNTER_FUKUDA_B AT %IB07 :	BYTE;
G6_ERROR1  AT %IB08 :	BYTE;
G6_ERROR2  AT %IB09 :	BYTE;
G6_OUTPUT AT %QB00 : 	BYTE;
G6_OUTPUT_1 AT %QB01 : BYTE;
G6_OUTPUT_2 AT %QB02 : BYTE;
START_POSITION AT %QB03 : BYTE :=1;

I_CMDERROR AT %IX09.6 :BOOL;
I_G6_READY  AT %IX0.0 :BOOL;
I_G6_RUNNING  AT %IX0.1 :BOOL;
I_G6_PAUSED  AT %IX0.2 :BOOL;
I_G6_ERROR  AT %IX0.3 :BOOL;
I_G6_ESTOPON  AT %IX0.4 :BOOL;
I_G6_SAFEGUARDON  AT %IX0.5 :BOOL;
I_G6_SERROR  AT %IX0.6 :BOOL;
I_G6_WARNING  AT %IX0.7 :BOOL;

I_G6_MOTORON  AT %IX1.0 :BOOL;
I_G6_ATHOME  AT %IX1.1 :BOOL;
I_G6_AUTOMODE  AT %IX1.5 :BOOL;
	
I_G6_END_CYCLE  AT %IX3.0 :BOOL;
I_G6_END_FUKUDA  AT %IX3.1 :BOOL;
I_G6_READY_TAKEUP  AT %IX3.2 :BOOL;//CYCLE RUNNING INDICATOR
I_G6_START_TAKEUP  AT %IX3.3 :BOOL;
I_G6_READY_PLACING  AT %IX3.4 :BOOL;
I_G6_START_PLACING  AT %IX3.5 :BOOL;
I_READY_CONTINUE  :BOOL;


	
	O_G6_START AT %QX00.0  : BOOL;	
	O_G6_SELECT_FUKUDA_A AT %QX00.1  : BOOL;
	O_G6_SELECT_FUKUDA_B AT %QX00.2  : BOOL;
	O_G6_STOP AT %QX00.4  : BOOL;
	O_G6_PAUSE AT %QX00.5  : BOOL;

	O_G6_RESET AT %QX00.7  : BOOL;	
	
	O_G6_SETMOTORON AT %QX01.0  : BOOL;
	O_G6_SETMOTOROFF AT %QX01.1  : BOOL;
	O_G6_HOME AT %QX01.2  : BOOL;
	O_G6_RESET_COUNTER_PICK AT %QX01.5  : BOOL:=FALSE;
	O_G6_CONTINUE AT %QX01.6  : BOOL;
	
I_G6_GRIPPER_CLOSE_1 AT %I* : BOOL;
I_G6_GRIPPER_CLOSE_2 AT %I* : BOOL;
I_G6_GRIPPER_CLOSE_3 AT %I* : BOOL;
I_G6_GRIPPER_CLOSE_4 AT %I* : BOOL;
I_G6_GRIPPER_OPEN_1 AT %I* : BOOL;
I_G6_GRIPPER_OPEN_2 AT %I* : BOOL;
I_G6_GRIPPER_OPEN_3 AT %I* : BOOL;
I_G6_GRIPPER_OPEN_4 AT %I* : BOOL;
I_G6_GRIPPER_EXT_DOWN_1 AT %I* : BOOL;
I_G6_GRIPPER_EXT_DOWN_2 AT %I* : BOOL;
I_G6_GRIPPER_EXT_DOWN_3 AT %I* : BOOL;
I_G6_GRIPPER_EXT_DOWN_4 AT %I* : BOOL;
I_G6_GRIPPER_EXT_UP_1 AT %I* : BOOL;
I_G6_GRIPPER_EXT_UP_2 AT %I* : BOOL;
I_G6_GRIPPER_EXT_UP_3 AT %I* : BOOL;
I_G6_GRIPPER_EXT_UP_4 AT %I* : BOOL;

	O_G6_GRIPPER_CLOSE_1 AT %Q* : BOOL;
	O_G6_GRIPPER_CLOSE_2 AT %Q* : BOOL;
	O_G6_GRIPPER_CLOSE_3 AT %Q* : BOOL;
	O_G6_GRIPPER_CLOSE_4 AT %Q* : BOOL;
	O_G6_GRIPPER_OPEN_1 AT %Q* : BOOL;
	O_G6_GRIPPER_OPEN_2 AT %Q* : BOOL;
	O_G6_GRIPPER_OPEN_3 AT %Q* : BOOL;
	O_G6_GRIPPER_OPEN_4 AT %Q* : BOOL;
	O_G6_GRIPPER_EXT_DOWN_1 AT %Q* : BOOL;
	O_G6_GRIPPER_EXT_DOWN_2 AT %Q* : BOOL;
	O_G6_GRIPPER_EXT_DOWN_3 AT %Q* : BOOL;
	O_G6_GRIPPER_EXT_DOWN_4 AT %Q* : BOOL;
	O_G6_GRIPPER_EXT_UP_1 AT %Q* : BOOL;
	O_G6_GRIPPER_EXT_UP_2 AT %Q* : BOOL;
	O_G6_GRIPPER_EXT_UP_3 AT %Q* : BOOL;
	O_G6_GRIPPER_EXT_UP_4 AT %Q* : BOOL;

IX_G6_GRIPPER_1 AT %IX2.0 : BOOL;
IX_G6_GRIPPER_2 AT %IX2.1 : BOOL;
IX_G6_GRIPPER_3 AT %IX2.2 : BOOL;
IX_G6_GRIPPER_4 AT %IX2.3 : BOOL;

IX_G6_GRIPPER_EXT_1 AT %IX2.4 : BOOL;
IX_G6_GRIPPER_EXT_2 AT %IX2.5 : BOOL;
IX_G6_GRIPPER_EXT_3 AT %IX2.6 : BOOL;
IX_G6_GRIPPER_EXT_4 AT %IX2.7 : BOOL;
(*
	OX_G6_GRIPPER_1 AT %QX02.0 : BOOL;
	OX_G6_GRIPPER_2 AT %QX02.1 : BOOL;
	OX_G6_GRIPPER_3 AT %QX02.2 : BOOL;
	OX_G6_GRIPPER_4 AT %QX02.3 : BOOL;

	OX_G6_GRIPPER_EXT_1 AT %QX02.4 : BOOL;
	OX_G6_GRIPPER_EXT_2 AT %QX02.5 : BOOL;
	OX_G6_GRIPPER_EXT_3 AT %QX02.6 : BOOL;
	OX_G6_GRIPPER_EXT_4 AT %QX02.7 : BOOL;
*)
GRIPPER_OPEN_1 AT %QX02.0 : BOOL;
GRIPPER_CLOSE_1 AT %QX02.1 : BOOL;
GRIPPER_OPEN_2 AT %QX02.2 : BOOL;
GRIPPER_CLOSE_2 AT %QX02.3 : BOOL;
GRIPPER_OPEN_3 AT %QX02.4 : BOOL;
GRIPPER_CLOSE_3 AT %QX02.5 : BOOL;
GRIPPER_OPEN_4 AT %QX02.6 : BOOL;
GRIPPER_CLOSE_4 AT %QX02.7 : BOOL;
IX_G6_FINISH AT %I* : BOOL;
I_G6_HANG : BOOL;
I_G6_ENABLE :BOOL;
I_G6_DISABLE :BOOL;
GO_ROBOT :BOOL;
I_MAX_DEVICE:BYTE:=80;
		
END_VAR

// ---- GVLs/INPUT_VAR.TcGVL
{attribute 'qualified_only'}
VAR_GLOBAL
I_LOTBOX_CLAMP_ON_1 AT %I* : BOOL;
I_LOTBOX_CLAMP_ON_2 AT %I* : BOOL;
I_LOTBOX_CLAMP_ON_3 AT %I* : BOOL;
I_LOTBOX_CLAMP_ON_4 AT %I* : BOOL;
I_LOTBOX_CLAMP_OFF_1 AT %I* : BOOL;
I_LOTBOX_CLAMP_OFF_2 AT %I* : BOOL;
I_LOTBOX_CLAMP_OFF_3 AT %I* : BOOL;
I_LOTBOX_CLAMP_OFF_4 AT %I* : BOOL;
	
I_LOTBOX_DETECT_1 AT %I* : BOOL;//LOTBOX_FUKUDA1_DETECT
I_LOTBOX_DETECT_2 AT %I* : BOOL;//LOTBOX_FUKUDA2_DETECT
I_LOTBOX_DETECT_3 AT %I* : BOOL;//LOTBOX_FUKUDA3_DETECT
I_LOTBOX_DETECT_4 AT %I* : BOOL;//LOTBOX_FUKUDA4_DETECT

I_VACUUM_ON AT %I* : BOOL;
I_VACUUM_OFF AT %I* : BOOL;

I_FUKUDA_TRANSFER_AT_FRONT_A AT %I* : BOOL;
I_FUKUDA_TRANSFER_AT_BACK_A AT %I* : BOOL;
I_FUKUDA_TRANSFER_AT_FRONT_B AT %I* : BOOL;
I_FUKUDA_TRANSFER_AT_BACK_B AT %I* : BOOL;
I_FUKUDA_TRANSFER_A_PICKING : BYTE:=1;
I_FUKUDA_TRANSFER_A_PICK_DONE : BOOL;
I_FUKUDA_TRANSFER_B_PICK_DONE : BOOL;
I_FUKUDA_TRANSFER_AT_A : BOOL;
I_FUKUDA_TRANSFER_AT_B : BOOL;

I_LOADING_SOCKET : T_JIG_SOCKET;
I_CURRENT_TRANSACTION : T_CURRENT_TRANSACTION ;
I_RETURN_DONE_A: BOOL;
I_RETURN_DONE_B: BOOL;
I_LOADING_DONE_A: BOOL;
I_LOADING_DONE_B: BOOL;
I_FUKUDA_ONDUTY_A:BOOL;
I_FUKUDA_ONDUTY_B:BOOL;
JIG_FUKUDA_PRESENCE: BOOL :=TRUE;

I_LOTEND :BOOL :=TRUE;
I_FUNC_CALLED:BOOL:=TRUE;
I_LOADING_DONE : BOOL;
I_LOADING_FAILED: BOOL;
I_LOADING_ALARM: INT;
I_CARTESSIAN_GRIPPER_ON AT %I* : BOOL;
I_CARTESSIAN_GRIPPER_OFF AT %I* : BOOL;
I_FUNCTION_NAME :STRING [255];
I_CASE : INT:=0;
I_FUKUDA_RUNNING:BOOL :=FALSE;

O_LOTBOX_CLAMP_ON_1 AT %Q* : BOOL;
O_LOTBOX_CLAMP_ON_2 AT %Q* : BOOL;
O_LOTBOX_CLAMP_ON_3 AT %Q* : BOOL;
O_LOTBOX_CLAMP_ON_4 AT %Q* : BOOL;
O_LOTBOX_CLAMP_OFF_1 AT %Q* : BOOL;
O_LOTBOX_CLAMP_OFF_2 AT %Q* : BOOL;
O_LOTBOX_CLAMP_OFF_3 AT %Q* : BOOL;
O_LOTBOX_CLAMP_OFF_4 AT %Q* : BOOL;

O_VACUUM_ON AT %Q* : BOOL;
O_VACUUM_OFF AT %Q* : BOOL;
O_CARTESSIAN_GRIPPER_ON AT %Q* : BOOL;
O_CARTESSIAN_GRIPPER_OFF AT %Q* : BOOL;
O_TOWER_LAMP_RED AT %Q* : BOOL;
O_TOWER_LAMP_YELLOW AT %Q* : BOOL;
O_TOWER_LAMP_GREEN AT %Q* : BOOL;
O_TOWER_LAMP_BUZZER AT %Q* : BOOL;
O_WARNING_LIGHT AT %Q* : BOOL;
O_LOT_BOX_INDICATOR_1  AT %Q* : BOOL;
O_LOT_BOX_INDICATOR_2 AT %Q* : BOOL;
O_LOT_BOX_INDICATOR_3 AT %Q* : BOOL;
O_LOT_BOX_INDICATOR_4 AT %Q* : BOOL;

AXIS_COMPLETE: BOOL;
LOTBOX_READY_1: BOOL;

DataWordInput1 AT %IB100 : ARRAY [0..15] OF WORD; 
DataWordInput2 AT %IB132 : ARRAY [16..31] OF WORD; 
DataWordInput3 AT %IB164 : ARRAY [32..47] OF WORD; 
DataWordInput4 AT %IB196 : ARRAY [48..56] OF WORD; 
DataWordOutput1 AT %QB100 : ARRAY [0..15] OF WORD; 
DataWordOutput2 AT %QB132 : ARRAY [16..31] OF WORD; 
DataWordOutput3 AT %QB164 : ARRAY [32..47] OF WORD; 
DataWordOutput4 AT %QB196 : ARRAY [48..56] OF WORD; 

I_RETURN_ALARM: INT;
I_RETURN_FAILED: BOOL;
ACTIVE_ID: INT :=1;	
ACTIVE_PROGRAM: INT ;
ACTIVE_PROGRAM_CHANGE:BOOL;
	
I_FUKUDA_HOME : BOOL;
O_FUKUDA_HOME : BOOL; 
STRAIGHTEN_START: BOOL;
STRAIGHTEN_PROCESS: BOOL;
STRAIGHTEN_DONE: BOOL;

FUKUDA_HOME: BOOL;

O_STOPPER_TRANSFER_A AT %Q* : BOOL;
O_STOPPER_TRANSFER_B AT %Q* : BOOL;
I_STOPPER_TRANSFER_ON_A AT %Q* : BOOL;
I_STOPPER_TRANSFER_OFF_A AT %Q* : BOOL;
I_STOPPER_TRANSFER_ON_B AT %Q* : BOOL;
I_STOPPER_TRANSFER_OFF_B AT %Q* : BOOL;
O_RESET_CARTESSIAN AT %Q* : BOOL;

TRANSPORT_IDX:BYTE;
STATION_LOAD_IDX:BYTE;
JIG_LOAD_IDX :BYTE;
STATION_RETURN_IDX:BYTE;
JIG_RETURN_IDX :BYTE;

ALARM1:BOOL;
ERROR_CODE:INT;
END_VAR

// ---- GVLs/LOADER_RS4_VAR.TcGVL



{attribute 'qualified_only'}
VAR_GLOBAL

LOADER_RS4_INPUT AT %IB32 : ARRAY [0..15] OF WORD; 
LOADER_RS4_INPUT_1 AT %IB33 : ARRAY [0..15] OF WORD;
LOADER_RS4_INPUT_2 AT %IB36 : ARRAY [0..15] OF WORD;
LOADER_RS4_INPUT_3 AT %IB37 : ARRAY [0..15] OF WORD;
LOADER_RS4_OUTPUT AT %QB32 : BYTE;
LOADER_RS4_OUTPUT_1 AT %QB33 : BYTE;

CARRIER_INDEX AT %QB38 : BYTE :=1;
LOADER_RS4_OUTPUT_2 AT %QB39 : BYTE;

GRIPPER_SENSOR AT %QB40: BYTE;
GRP_SENS_OPEN_1 AT %QX40.0 : BOOL;
GRP_SENS_CLOSE_1 AT %QX40.1 : BOOL;
GRP_SENS_OPEN_2 AT %QX40.2: BOOL;
GRP_SENS_CLOSE_2 AT %QX40.3 : BOOL;
GRP_SENS_OPEN_3 AT %QX40.4: BOOL;
GRP_SENS_CLOSE_3 AT %QX40.5 : BOOL;
GRP_SENS_OPEN_4 AT %QX40.6: BOOL;
GRP_SENS_CLOSE_4 AT %QX40.7 : BOOL;

O_END_CARRIER AT %QX39.0 : BOOL;
I_LOADER_RS4_READY  AT %IX32.0 :BOOL;
I_LOADER_RS4_RUNNING  AT %IX32.1 :BOOL;
I_LOADER_RS4_PAUSED  AT %IX32.2 :BOOL;
I_LOADER_RS4_ERROR  AT %IX32.3 :BOOL;
I_LOADER_RS4_ESTOPON  AT %IX32.4 :BOOL;
I_LOADER_RS4_SAFEGUARDON  AT %IX32.5 :BOOL;
I_LOADER_RS4_SERROR  AT %IX32.6 :BOOL;
I_LOADER_RS4_WARNING  AT %IX32.7 :BOOL;

I_LOADER_RS4_MOTORON  AT %IX33.0 :BOOL;
I_LOADER_RS4_ATHOME  AT %IX33.1 :BOOL;
I_LOADER_RS4_AUTOMODE  AT %IX33.5 :BOOL;
	
I_LOADER_RS4_END_CYCLE  AT %IX37.0 :BOOL;
I_LOADER_RS4_END_FUKUDA  AT %IX37.1 :BOOL;
I_LOADER_RS4_END_CARRIER :BOOL;
POSITION_TOOL_1 AT %QB34 : BYTE :=0;
POSITION_TOOL_2 AT %QB35 : BYTE :=0;
POSITION_TOOL_3 AT %QB36 : BYTE :=1;
POSITION_TOOL_4 AT %QB37 : BYTE :=2;
I_LOADER_RS4_ENABLE :BOOL ;
I_LOADER_RS4_READY_TAKEUP  AT %IX37.2 :BOOL;//CYCLE RUNNING INDICATOR
I_LOADER_RS4_START_TAKEUP  AT %IX37.3 :BOOL;
I_LOADER_RS4_READY_PLACING  AT %IX37.4 :BOOL;
I_LOADER_RS4_START_PLACING  AT %IX37.5 :BOOL;
	
	O_LOADER_RS4_START AT %QX32.0  : BOOL;	
	O_LOADER_RS4_SELECT_FUKUDA_A AT %QX32.1  : BOOL;
	O_LOADER_RS4_SELECT_FUKUDA_B AT %QX32.2  : BOOL;
	O_LOADER_RS4_STOP AT %QX32.4  : BOOL;
	O_LOADER_RS4_PAUSE AT %QX32.5  : BOOL;
	O_LOADER_RS4_CONTINUE AT %QX33.6  : BOOL;
	O_LOADER_RS4_RESET AT %QX32.7  : BOOL;	
	
	O_LOADER_RS4_SETMOTORON AT %QX33.0  : BOOL;
	O_LOADER_RS4_SETMOTOROFF AT %QX33.1  : BOOL;
	O_LOADER_RS4_HOME AT %QX33.2  : BOOL;

I_LOADER_RS4_GRIPPER_CLOSE_1 AT %I* : BOOL;
I_LOADER_RS4_GRIPPER_CLOSE_2 AT %I* : BOOL;
I_LOADER_RS4_GRIPPER_CLOSE_3 AT %I* : BOOL;
I_LOADER_RS4_GRIPPER_CLOSE_4 AT %I* : BOOL;
I_LOADER_RS4_GRIPPER_OPEN_1 AT %I* : BOOL;
I_LOADER_RS4_GRIPPER_OPEN_2 AT %I* : BOOL;
I_LOADER_RS4_GRIPPER_OPEN_3 AT %I* : BOOL;
I_LOADER_RS4_GRIPPER_OPEN_4 AT %I* : BOOL;
I_LOADER_RS4_GRIPPER_EXT_DOWN_1 AT %I* : BOOL;
I_LOADER_RS4_GRIPPER_EXT_DOWN_2 AT %I* : BOOL;
I_LOADER_RS4_GRIPPER_EXT_DOWN_3 AT %I* : BOOL;
I_LOADER_RS4_GRIPPER_EXT_DOWN_4 AT %I* : BOOL;
I_LOADER_RS4_GRIPPER_EXT_UP_1 AT %I* : BOOL;
I_LOADER_RS4_GRIPPER_EXT_UP_2 AT %I* : BOOL;
I_LOADER_RS4_GRIPPER_EXT_UP_3 AT %I* : BOOL;
I_LOADER_RS4_GRIPPER_EXT_UP_4 AT %I* : BOOL;

O_LOADER_RS4_GRIPPER_CLOSE_1 AT %Q* : BOOL;
O_LOADER_RS4_GRIPPER_CLOSE_2 AT %Q* : BOOL;
O_LOADER_RS4_GRIPPER_CLOSE_3 AT %Q* : BOOL;
O_LOADER_RS4_GRIPPER_CLOSE_4 AT %Q* : BOOL;
O_LOADER_RS4_GRIPPER_OPEN_1 AT %Q* : BOOL;
O_LOADER_RS4_GRIPPER_OPEN_2 AT %Q* : BOOL;
O_LOADER_RS4_GRIPPER_OPEN_3 AT %Q* : BOOL;
O_LOADER_RS4_GRIPPER_OPEN_4 AT %Q* : BOOL;
O_LOADER_RS4_GRIPPER_EXT_DOWN_1 AT %Q* : BOOL;
O_LOADER_RS4_GRIPPER_EXT_DOWN_2 AT %Q* : BOOL;
O_LOADER_RS4_GRIPPER_EXT_DOWN_3 AT %Q* : BOOL;
O_LOADER_RS4_GRIPPER_EXT_DOWN_4 AT %Q* : BOOL;
O_LOADER_RS4_GRIPPER_EXT_UP_1 AT %Q* : BOOL;
O_LOADER_RS4_GRIPPER_EXT_UP_2 AT %Q* : BOOL;
O_LOADER_RS4_GRIPPER_EXT_UP_3 AT %Q* : BOOL;
O_LOADER_RS4_GRIPPER_EXT_UP_4 AT %Q* : BOOL;

IX_LOADER_RS4_GRIPPER_1 AT %IX36.0 : BOOL;
IX_LOADER_RS4_GRIPPER_2 AT %IX36.1 : BOOL;
IX_LOADER_RS4_GRIPPER_3 AT %IX36.2 : BOOL;
IX_LOADER_RS4_GRIPPER_4 AT %IX36.3 : BOOL;

IX_LOADER_RS4_GRIPPER_EXT_1 AT %IX36.4 : BOOL;
IX_LOADER_RS4_GRIPPER_EXT_2 AT %IX36.5 : BOOL;
IX_LOADER_RS4_GRIPPER_EXT_3 AT %IX36.6 : BOOL;
IX_LOADER_RS4_GRIPPER_EXT_4 AT %IX36.7 : BOOL;


IX_LOADER_RS4_HOME AT %I* : BOOL;
IX_LOADER_RS4_RUNNING AT %I* : BOOL;
IX_LOADER_RS4_PICKUP_1 AT %I* : BOOL;
IX_LOADER_RS4_PICKUP_2 AT %I* : BOOL;
IX_LOADER_RS4_PICKUP_3 AT %I* : BOOL;
IX_LOADER_RS4_PICKUP_4 AT %I* : BOOL;
IX_LOADER_RS4_PLACING_1 AT %I* : BOOL;
IX_LOADER_RS4_PLACING_2 AT %I* : BOOL;
IX_LOADER_RS4_PLACING_3 AT %I* : BOOL;
IX_LOADER_RS4_PLACING_4 AT %I* : BOOL;

IX_LOADER_RS4_FINISH AT %I* : BOOL;
I_LOADER_RS4_HANG :BOOL;
I_LOADER_RS4_DISABLE :BOOL;
I_READY_CONTINUE : BOOL;
FINISH_POSITION_TOOL : INT;

READY_INDEXING :BOOL;

	
END_VAR

// ---- GVLs/LOADER_VAR.TcGVL
(*{attribute 'qualified_only'}
VAR_GLOBAL
I_LOADER_CLAMPING_ON_1 AT %I* : BOOL;
I_LOADER_CLAMPING_ON_2 AT %I* : BOOL;
I_LOADER_CLAMPING_ON_3 AT %I* : BOOL;
I_LOADER_CLAMPING_ON_4 AT %I* : BOOL;
I_LOADER_CLAMPING_OFF_1 AT %I* : BOOL;
I_LOADER_CLAMPING_OFF_2 AT %I* : BOOL;
I_LOADER_CLAMPING_OFF_3 AT %I* : BOOL;
I_LOADER_CLAMPING_OFF_4 AT %I* : BOOL;

I_CARRIER_DETECT_1 AT %I* : BOOL;
I_CARRIER_DETECT_2 AT %I* : BOOL;
I_CARRIER_DETECT_3 AT %I* : BOOL;
I_CARRIER_DETECT_4 AT %I* : BOOL;

I_C8_FRONT_LIMIT AT %I* : BOOL;
I_C8_REAR_LIMIT AT %I* : BOOL;
I_ENABLE_SWITCH AT %I* : BOOL;
I_DISABLE_SWITCH AT %I* : BOOL;
I_EMERGENCY_SWITCH AT %I* : BOOL;
I_SAFETY_CURTAIN_1 AT %I* : BOOL;
I_SAFETY_CURTAIN_2 AT %I* : BOOL;
I_BUYOFF_RACK_1 AT %I* : BOOL;
I_BUYOFF_RACK_2 AT %I* : BOOL;
I_BUYOFF_RACK_3 AT %I* : BOOL;
I_BUYOFF_RACK_4 AT %I* : BOOL;
I_BUYOFF_RACK_5 AT %I* : BOOL;
I_BUYOFF_RACK_6 AT %I* : BOOL;
I_BUYOFF_RACK_7 AT %I* : BOOL;
I_BUYOFF_RACK_8 AT %I* : BOOL;
I_BUYOFF_RACK_9 AT %I* : BOOL;
I_BUYOFF_RACK_10 AT %I* : BOOL;
I_BUYOFF_RACK_11 AT %I* : BOOL;
I_BUYOFF_RACK_12 AT %I* : BOOL;
I_BUYOFF_RACK_13 AT %I* : BOOL;
I_BUYOFF_RACK_14 AT %I* : BOOL;
I_BUYOFF_RACK_15 AT %I* : BOOL;
I_BUYOFF_RACK_16 AT %I* : BOOL;
I_BUYOFF_RACK_17 AT %I* : BOOL;
I_BUYOFF_RACK_18 AT %I* : BOOL;
I_BUYOFF_RACK_19 AT %I* : BOOL;
I_BUYOFF_RACK_20 AT %I* : BOOL;
I_BUYOFF_RACK_21 AT %I* : BOOL;
I_BUYOFF_RACK_22 AT %I* : BOOL;
I_BUYOFF_RACK_23 AT %I* : BOOL;
I_BUYOFF_RACK_24 AT %I* : BOOL;
I_C8_GRIPPER_ON AT %I* : BOOL;
I_C8_GRIPPER_OFF AT %I* : BOOL;
I_SAFETY_FENCE_OPEN_1 AT %I* : BOOL;
I_SAFETY_FENCE_OPEN_2 AT %I* : BOOL;
I_SAFETY_FENCE_OPEN_3 AT %I* : BOOL;
I_SAFETY_FENCE_OPEN_4 AT %I* : BOOL;
I_SAFETY_FENCE_OPEN_5 AT %I* : BOOL;
I_SAFETY_FENCE_OPEN_6 AT %I* : BOOL;
I_SAFETY_FENCE_OPEN_7 AT %I* : BOOL;
I_SAFETY_FENCE_OPEN_8 AT %I* : BOOL;
I_SAFETY_FENCE_OPEN_9 AT %I* : BOOL;
I_SAFETY_FENCE_OPEN_10 AT %I* : BOOL;
I_SAFETY_FENCE_OPEN_11 AT %I* : BOOL;
I_SAFETY_FENCE_OPEN_12 AT %I* : BOOL;
I_SAFETY_FENCE_LOCK_ON_1 AT %I* : BOOL;
I_SAFETY_FENCE_LOCK_ON_2 AT %I* : BOOL;
I_SAFETY_FENCE_LOCK_ON_3 AT %I* : BOOL;
I_SAFETY_FENCE_LOCK_ON_4 AT %I* : BOOL;
I_SAFETY_FENCE_LOCK_ON_5 AT %I* : BOOL;
I_SAFETY_FENCE_LOCK_ON_6 AT %I* : BOOL;
I_SAFETY_FENCE_LOCK_ON_7 AT %I* : BOOL;
I_SAFETY_FENCE_LOCK_ON_8 AT %I* : BOOL;
I_SAFETY_FENCE_LOCK_ON_9 AT %I* : BOOL;
I_SAFETY_FENCE_LOCK_ON_10 AT %I* : BOOL;
I_SAFETY_FENCE_LOCK_ON_11 AT %I* : BOOL;
I_SAFETY_FENCE_LOCK_ON_12 AT %I* : BOOL;
I_SAFETY_FENCE_LOCK_OFF_1 AT %I* : BOOL;
I_SAFETY_FENCE_LOCK_OFF_2 AT %I* : BOOL;
I_SAFETY_FENCE_LOCK_OFF_3 AT %I* : BOOL;
I_SAFETY_FENCE_LOCK_OFF_4 AT %I* : BOOL;
I_SAFETY_FENCE_LOCK_OFF_5 AT %I* : BOOL;
I_SAFETY_FENCE_LOCK_OFF_6 AT %I* : BOOL;
I_SAFETY_FENCE_LOCK_OFF_7 AT %I* : BOOL;
I_SAFETY_FENCE_LOCK_OFF_8 AT %I* : BOOL;
I_SAFETY_FENCE_LOCK_OFF_9 AT %I* : BOOL;
I_SAFETY_FENCE_LOCK_OFF_10 AT %I* : BOOL;
I_SAFETY_FENCE_LOCK_OFF_11 AT %I* : BOOL;
I_SAFETY_FENCE_LOCK_OFF_12 AT %I* : BOOL;
I_TESTER_NOISE_ENABLE_1 AT %I* : BOOL;
I_TESTER_NOISE_ENABLE_2 AT %I* : BOOL;
I_TESTER_NOISE_ENABLE_3 AT %I* : BOOL;
I_TESTER_NOISE_ENABLE_4 AT %I* : BOOL;
I_TESTER_NOISE_ENABLE_5 AT %I* : BOOL;
I_TESTER_NOISE_ENABLE_6 AT %I* : BOOL;
I_TESTER_NOISE_ENABLE_7 AT %I* : BOOL;
I_TESTER_NOISE_ENABLE_8 AT %I* : BOOL;
I_TESTER_SIGNAL_ENABLE_1 AT %I* : BOOL;
I_TESTER_SIGNAL_ENABLE_2 AT %I* : BOOL;
I_TESTER_RESISTANCE_ENABLE_1 AT %I* : BOOL;
I_TESTER_RESISTANCE_ENABLE_2 AT %I* : BOOL;
I_TESTER_NOISE_DISABLE_1 AT %I* : BOOL;
I_TESTER_NOISE_DISABLE_2 AT %I* : BOOL;
I_TESTER_NOISE_DISABLE_3 AT %I* : BOOL;
I_TESTER_NOISE_DISABLE_4 AT %I* : BOOL;
I_TESTER_NOISE_DISABLE_5 AT %I* : BOOL;
I_TESTER_NOISE_DISABLE_6 AT %I* : BOOL;
I_TESTER_NOISE_DISABLE_7 AT %I* : BOOL;
I_TESTER_NOISE_DISABLE_8 AT %I* : BOOL;
I_TESTER_SIGNAL_DISABLE_1 AT %I* : BOOL;
I_TESTER_SIGNAL_DISABLE_2 AT %I* : BOOL;
I_TESTER_RESISTANCE_DISABLE_1 AT %I* : BOOL;
I_TESTER_RESISTANCE_DISABLE_2 AT %I* : BOOL;
I_TESTER_NOISE_EMERGENCY_1 AT %I* : BOOL;
I_TESTER_NOISE_EMERGENCY_2 AT %I* : BOOL;
I_TESTER_NOISE_EMERGENCY_3 AT %I* : BOOL;
I_TESTER_NOISE_EMERGENCY_4 AT %I* : BOOL;
I_TESTER_NOISE_EMERGENCY_5 AT %I* : BOOL;
I_TESTER_NOISE_EMERGENCY_6 AT %I* : BOOL;
I_TESTER_NOISE_EMERGENCY_7 AT %I* : BOOL;
I_TESTER_NOISE_EMERGENCY_8 AT %I* : BOOL;
I_TESTER_SIGNAL_EMERGENCY_1 AT %I* : BOOL;
I_TESTER_SIGNAL_EMERGENCY_2 AT %I* : BOOL;
I_TESTER_RESISTANCE_EMERGENCY_1 AT %I* : BOOL;
I_TESTER_RESISTANCE_EMERGENCY_2 AT %I* : BOOL;
I_BUFFER_CARRIER_DETECT_1 AT %I* : BOOL;
I_BUFFER_CARRIER_DETECT_2 AT %I* : BOOL;
I_INPUT_CARTESSIAN_HOME AT %I* : BOOL;
I_INPUT_CARTESSIAN_RUNNING AT %I* : BOOL;
I_INPUT_CARTESSIAN_FINISH AT %I* : BOOL;
I_TESTER_READY_1 AT %I* : BOOL;
I_TESTER_READY_2 AT %I* : BOOL;
I_TESTER_READY_3 AT %I* : BOOL;
I_TESTER_READY_4 AT %I* : BOOL;
I_TESTER_READY_5 AT %I* : BOOL;
I_TESTER_READY_6 AT %I* : BOOL;
I_TESTER_READY_7 AT %I* : BOOL;
I_TESTER_READY_8 AT %I* : BOOL;
I_TESTER_READY_9 AT %I* : BOOL;
I_TESTER_READY_10 AT %I* : BOOL;
I_TESTER_READY_11 AT %I* : BOOL;
I_TESTER_READY_12 AT %I* : BOOL;

O_LOADER_CLAMPING_ON_1 AT %Q* : BOOL;
O_LOADER_CLAMPING_ON_2 AT %Q* : BOOL;
O_LOADER_CLAMPING_ON_3 AT %Q* : BOOL;
O_LOADER_CLAMPING_ON_4 AT %Q* : BOOL;
O_LOADER_CLAMPING_OFF_1 AT %Q* : BOOL;
O_LOADER_CLAMPING_OFF_2 AT %Q* : BOOL;
O_LOADER_CLAMPING_OFF_3 AT %Q* : BOOL;
O_LOADER_CLAMPING_OFF_4 AT %Q* : BOOL;
O_C8_GRIPPER_ON AT %Q* : BOOL;
O_C8_GRIPPER_OFF AT %Q* : BOOL;
O_SAFETY_FENCE_NOISE_LOCK_ON_1 AT %Q* : BOOL;
O_SAFETY_FENCE_NOISE_LOCK_ON_2 AT %Q* : BOOL;
O_SAFETY_FENCE_NOISE_LOCK_ON_3 AT %Q* : BOOL;
O_SAFETY_FENCE_NOISE_LOCK_ON_4 AT %Q* : BOOL;
O_SAFETY_FENCE_NOISE_LOCK_ON_5 AT %Q* : BOOL;
O_SAFETY_FENCE_NOISE_LOCK_ON_6 AT %Q* : BOOL;
O_SAFETY_FENCE_NOISE_LOCK_ON_7 AT %Q* : BOOL;
O_SAFETY_FENCE_NOISE_LOCK_ON_8 AT %Q* : BOOL;
O_SAFETY_FENCE_SIGNAL_LOCK_ON_1 AT %Q* : BOOL;
O_SAFETY_FENCE_SIGNAL_LOCK_ON_2 AT %Q* : BOOL;
O_SAFETY_FENCE_RESISTANCE_LOCK_ON_1 AT %Q* : BOOL;
O_SAFETY_FENCE_RESISTANCE_LOCK_ON_2 AT %Q* : BOOL;
O_TESTER_TOWER_NOISE_LAMP_RED_1 AT %Q* : BOOL;
O_TESTER_TOWER_NOISE_LAMP_RED_2 AT %Q* : BOOL;
O_TESTER_TOWER_NOISE_LAMP_RED_3 AT %Q* : BOOL;
O_TESTER_TOWER_NOISE_LAMP_RED_4 AT %Q* : BOOL;
O_TESTER_TOWER_NOISE_LAMP_RED_5 AT %Q* : BOOL;
O_TESTER_TOWER_NOISE_LAMP_RED_6 AT %Q* : BOOL;
O_TESTER_TOWER_NOISE_LAMP_RED_7 AT %Q* : BOOL;
O_TESTER_TOWER_NOISE_LAMP_RED_8 AT %Q* : BOOL;
O_TESTER_TOWER_SIGNAL_LAMP_RED_1 AT %Q* : BOOL;
O_TESTER_TOWER_SIGNAL_LAMP_RED_2 AT %Q* : BOOL;
O_TESTER_TOWER_RESISTANCE_LAMP_RED_1 AT %Q* : BOOL;
O_TESTER_TOWER_RESISTANCE_LAMP_RED_2 AT %Q* : BOOL;
O_TESTER_TOWER_NOISE_LAMP_YELLOW_1 AT %Q* : BOOL;
O_TESTER_TOWER_NOISE_LAMP_YELLOW_2 AT %Q* : BOOL;
O_TESTER_TOWER_NOISE_LAMP_YELLOW_3 AT %Q* : BOOL;
O_TESTER_TOWER_NOISE_LAMP_YELLOW_4 AT %Q* : BOOL;
O_TESTER_TOWER_NOISE_LAMP_YELLOW_5 AT %Q* : BOOL;
O_TESTER_TOWER_NOISE_LAMP_YELLOW_6 AT %Q* : BOOL;
O_TESTER_TOWER_NOISE_LAMP_YELLOW_7 AT %Q* : BOOL;
O_TESTER_TOWER_NOISE_LAMP_YELLOW_8 AT %Q* : BOOL;
O_TESTER_TOWER_SIGNAL_LAMP_YELLOW_1 AT %Q* : BOOL;
O_TESTER_TOWER_SIGNAL_LAMP_YELLOW_2 AT %Q* : BOOL;
O_TESTER_TOWER_RESISTANCE_LAMP_YELLOW_1 AT %Q* : BOOL;
O_TESTER_TOWER_RESISTANCE_LAMP_YELLOW_2 AT %Q* : BOOL;
O_TESTER_TOWER_NOISE_LAMP_GREEN_1 AT %Q* : BOOL;
O_TESTER_TOWER_NOISE_LAMP_GREEN_2 AT %Q* : BOOL;
O_TESTER_TOWER_NOISE_LAMP_GREEN_3 AT %Q* : BOOL;
O_TESTER_TOWER_NOISE_LAMP_GREEN_4 AT %Q* : BOOL;
O_TESTER_TOWER_NOISE_LAMP_GREEN_5 AT %Q* : BOOL;
O_TESTER_TOWER_NOISE_LAMP_GREEN_6 AT %Q* : BOOL;
O_TESTER_TOWER_NOISE_LAMP_GREEN_7 AT %Q* : BOOL;
O_TESTER_TOWER_NOISE_LAMP_GREEN_8 AT %Q* : BOOL;
O_TESTER_TOWER_SIGNAL_LAMP_GREEN_1 AT %Q* : BOOL;
O_TESTER_TOWER_SIGNAL_LAMP_GREEN_2 AT %Q* : BOOL;
O_TESTER_TOWER_RESISTANCE_LAMP_GREEN_1 AT %Q* : BOOL;
O_TESTER_TOWER_RESISTANCE_LAMP_GREEN_2 AT %Q* : BOOL;
O_TESTER_CHILLER_NOISE_ON_1 AT %Q* : BOOL;
O_TESTER_CHILLER_NOISE_ON_2 AT %Q* : BOOL;
O_TESTER_CHILLER_NOISE_ON_3 AT %Q* : BOOL;
O_TESTER_CHILLER_NOISE_ON_4 AT %Q* : BOOL;
O_TESTER_CHILLER_NOISE_ON_5 AT %Q* : BOOL;
O_TESTER_CHILLER_NOISE_ON_6 AT %Q* : BOOL;
O_TESTER_CHILLER_NOISE_ON_7 AT %Q* : BOOL;
O_TESTER_CHILLER_NOISE_ON_8 AT %Q* : BOOL;
O_TESTER_CHILLER_SIGNAL_ON_1 AT %Q* : BOOL;
O_TESTER_CHILLER_SIGNAL_ON_2 AT %Q* : BOOL;
O_TESTER_CHILLER_RESISTANCE_ON_1 AT %Q* : BOOL;
O_TESTER_CHILLER_RESISTANCE_ON_2 AT %Q* : BOOL;
O_TESTER_CHILLER_NOISE_OFF_1 AT %Q* : BOOL;
O_TESTER_CHILLER_NOISE_OFF_2 AT %Q* : BOOL;
O_TESTER_CHILLER_NOISE_OFF_3 AT %Q* : BOOL;
O_TESTER_CHILLER_NOISE_OFF_4 AT %Q* : BOOL;
O_TESTER_CHILLER_NOISE_OFF_5 AT %Q* : BOOL;
O_TESTER_CHILLER_NOISE_OFF_6 AT %Q* : BOOL;
O_TESTER_CHILLER_NOISE_OFF_7 AT %Q* : BOOL;
O_TESTER_CHILLER_NOISE_OFF_8 AT %Q* : BOOL;
O_TESTER_CHILLER_SIGNAL_OFF_1 AT %Q* : BOOL;
O_TESTER_CHILLER_SIGNAL_OFF_2 AT %Q* : BOOL;
O_TESTER_CHILLER_RESISTANCE_OFF_1 AT %Q* : BOOL;
O_TESTER_CHILLER_RESISTANCE_OFF_2 AT %Q* : BOOL;
O_TESTER_POWER_NOISE_ON_1 AT %Q* : BOOL;
O_TESTER_POWER_NOISE_ON_2 AT %Q* : BOOL;
O_TESTER_POWER_NOISE_ON_3 AT %Q* : BOOL;
O_TESTER_POWER_NOISE_ON_4 AT %Q* : BOOL;
O_TESTER_POWER_NOISE_ON_5 AT %Q* : BOOL;
O_TESTER_POWER_NOISE_ON_6 AT %Q* : BOOL;
O_TESTER_POWER_NOISE_ON_7 AT %Q* : BOOL;
O_TESTER_POWER_NOISE_ON_8 AT %Q* : BOOL;
O_TESTER_POWER_SIGNAL_ON_1 AT %Q* : BOOL;
O_TESTER_POWER_SIGNAL_ON_2 AT %Q* : BOOL;
O_TESTER_POWER_RESISTANCE_ON_1 AT %Q* : BOOL;
O_TESTER_POWER_RESISTANCE_ON_2 AT %Q* : BOOL;
O_TESTER_PC_SWITCH_NOISE_ON_1 AT %Q* : BOOL;
O_TESTER_PC_SWITCH_NOISE_ON_2 AT %Q* : BOOL;
O_TESTER_PC_SWITCH_NOISE_ON_3 AT %Q* : BOOL;
O_TESTER_PC_SWITCH_NOISE_ON_4 AT %Q* : BOOL;
O_TESTER_PC_SWITCH_NOISE_ON_5 AT %Q* : BOOL;
O_TESTER_PC_SWITCH_NOISE_ON_6 AT %Q* : BOOL;
O_TESTER_PC_SWITCH_NOISE_ON_7 AT %Q* : BOOL;
O_TESTER_PC_SWITCH_NOISE_ON_8 AT %Q* : BOOL;
O_TESTER_PC_SWITCH_SIGNAL_ON_1 AT %Q* : BOOL;
O_TESTER_PC_SWITCH_SIGNAL_ON_2 AT %Q* : BOOL;
O_TESTER_PC_SWITCH_RESISTANCE_ON_1 AT %Q* : BOOL;
O_TESTER_PC_SWITCH_RESISTANCE_ON_2 AT %Q* : BOOL;
O_TESTER_NOISE_START_1 AT %Q* : BOOL;
O_TESTER_NOISE_START_2 AT %Q* : BOOL;
O_TESTER_NOISE_START_3 AT %Q* : BOOL;
O_TESTER_NOISE_START_4 AT %Q* : BOOL;
O_TESTER_NOISE_START_5 AT %Q* : BOOL;
O_TESTER_NOISE_START_6 AT %Q* : BOOL;
O_TESTER_NOISE_START_7 AT %Q* : BOOL;
O_TESTER_NOISE_START_8 AT %Q* : BOOL;
O_TESTER_SIGNAL_START_1 AT %Q* : BOOL;
O_TESTER_SIGNAL_START_2 AT %Q* : BOOL;
O_TESTER_RESISTANCE_START_1 AT %Q* : BOOL;
O_TESTER_RESISTANCE_START_2 AT %Q* : BOOL;
O_TESTER_NOISE_STOP_1 AT %Q* : BOOL;
O_TESTER_NOISE_STOP_2 AT %Q* : BOOL;
O_TESTER_NOISE_STOP_3 AT %Q* : BOOL;
O_TESTER_NOISE_STOP_4 AT %Q* : BOOL;
O_TESTER_NOISE_STOP_5 AT %Q* : BOOL;
O_TESTER_NOISE_STOP_6 AT %Q* : BOOL;
O_TESTER_NOISE_STOP_7 AT %Q* : BOOL;
O_TESTER_NOISE_STOP_8 AT %Q* : BOOL;
O_TESTER_SIGNAL_STOP_1 AT %Q* : BOOL;
O_TESTER_SIGNAL_STOP_2 AT %Q* : BOOL;
O_TESTER_RESISTANCE_STOP_1 AT %Q* : BOOL;
O_TESTER_RESISTANCE_STOP_2 AT %Q* : BOOL;
O_TESTER_EMERGENCY_STOP_1 AT %Q* : BOOL;
O_TESTER_EMERGENCY_STOP_2 AT %Q* : BOOL;
O_TESTER_EMERGENCY_STOP_3 AT %Q* : BOOL;
O_TESTER_EMERGENCY_STOP_4 AT %Q* : BOOL;
O_TESTER_EMERGENCY_STOP_5 AT %Q* : BOOL;
O_TESTER_EMERGENCY_STOP_6 AT %Q* : BOOL;
O_TESTER_EMERGENCY_STOP_7 AT %Q* : BOOL;
O_TESTER_EMERGENCY_STOP_8 AT %Q* : BOOL;
O_TESTER_EMERGENCY_STOP_9 AT %Q* : BOOL;
O_TESTER_EMERGENCY_STOP_10 AT %Q* : BOOL;
O_TESTER_EMERGENCY_STOP_11 AT %Q* : BOOL;
O_TESTER_EMERGENCY_STOP_12 AT %Q* : BOOL;

I_TESTER_JIG_PRESENCE_1 AT %I* : BOOL;
I_TESTER_JIG_PRESENCE_2 AT %I* : BOOL;
I_TESTER_JIG_PRESENCE_3 AT %I* : BOOL;
I_TESTER_JIG_PRESENCE_4 AT %I* : BOOL;
I_TESTER_JIG_PRESENCE_5 AT %I* : BOOL;
I_TESTER_JIG_PRESENCE_6 AT %I* : BOOL;
I_TESTER_JIG_PRESENCE_7 AT %I* : BOOL;
I_TESTER_JIG_PRESENCE_8 AT %I* : BOOL;

END_VAR*)

{attribute 'qualified_only'}
VAR_GLOBAL
I_LOADER_CLAMPING_ON_1 AT %I* : BOOL;
I_LOADER_CLAMPING_ON_2 AT %I* : BOOL;
I_LOADER_CLAMPING_ON_3 AT %I* : BOOL;
I_LOADER_CLAMPING_ON_4 AT %I* : BOOL;
I_LOADER_CLAMPING_OFF_1 AT %I* : BOOL;
I_LOADER_CLAMPING_OFF_2 AT %I* : BOOL;
I_LOADER_CLAMPING_OFF_3 AT %I* : BOOL;
I_LOADER_CLAMPING_OFF_4 AT %I* : BOOL;

I_CARRIER_DETECT_1 AT %I* : BOOL;
I_CARRIER_DETECT_2 AT %I* : BOOL;
I_CARRIER_DETECT_3 AT %I* : BOOL;
I_CARRIER_DETECT_4 AT %I* : BOOL;

I_C8_FRONT_LIMIT AT %I* : BOOL;
I_C8_REAR_LIMIT AT %I* : BOOL;
I_ENABLE_SWITCH AT %I* : BOOL;
I_DISABLE_SWITCH AT %I* : BOOL;
I_EMERGENCY_SWITCH AT %I* : BOOL;
I_SAFETY_CURTAIN_1 AT %I* : BOOL;
I_SAFETY_CURTAIN_2 AT %I* : BOOL;
I_BUYOFF_RACK_1 AT %I* : BOOL;
I_BUYOFF_RACK_2 AT %I* : BOOL;
I_BUYOFF_RACK_3 AT %I* : BOOL;
I_BUYOFF_RACK_4 AT %I* : BOOL;
I_BUYOFF_RACK_5 AT %I* : BOOL;
I_BUYOFF_RACK_6 AT %I* : BOOL;
I_BUYOFF_RACK_7 AT %I* : BOOL;
I_BUYOFF_RACK_8 AT %I* : BOOL;
I_BUYOFF_RACK_9 AT %I* : BOOL;
I_BUYOFF_RACK_10 AT %I* : BOOL;
I_BUYOFF_RACK_11 AT %I* : BOOL;
I_BUYOFF_RACK_12 AT %I* : BOOL;
I_BUYOFF_RACK_13 AT %I* : BOOL;
I_BUYOFF_RACK_14 AT %I* : BOOL;
I_BUYOFF_RACK_15 AT %I* : BOOL;
I_BUYOFF_RACK_16 AT %I* : BOOL;
I_BUYOFF_RACK_17 AT %I* : BOOL;
I_BUYOFF_RACK_18 AT %I* : BOOL;
I_BUYOFF_RACK_19 AT %I* : BOOL;
I_BUYOFF_RACK_20 AT %I* : BOOL;
I_BUYOFF_RACK_21 AT %I* : BOOL;
I_BUYOFF_RACK_22 AT %I* : BOOL;
I_BUYOFF_RACK_23 AT %I* : BOOL;
I_BUYOFF_RACK_24 AT %I* : BOOL;
I_C8_GRIPPER_ON AT %I* : BOOL;
I_C8_GRIPPER_OFF AT %I* : BOOL;

//NOISE ROOM NUMBER : 11,12,13,14,15,16,17,18
//SIGNAL ROOM NUMBER : 21,22
//RESISTANCE ROOM NUMBER : 31,32
I_SAFETY_FENCE_OPEN_11 AT %I* : BOOL;
I_SAFETY_FENCE_OPEN_12 AT %I* : BOOL;
I_SAFETY_FENCE_OPEN_13 AT %I* : BOOL;
I_SAFETY_FENCE_OPEN_14 AT %I* : BOOL;
I_SAFETY_FENCE_OPEN_15 AT %I* : BOOL;
I_SAFETY_FENCE_OPEN_16 AT %I* : BOOL;
I_SAFETY_FENCE_OPEN_17 AT %I* : BOOL;
I_SAFETY_FENCE_OPEN_18 AT %I* : BOOL;
I_SAFETY_FENCE_OPEN_21 AT %I* : BOOL;
I_SAFETY_FENCE_OPEN_22 AT %I* : BOOL;
I_SAFETY_FENCE_OPEN_31 AT %I* : BOOL;
I_SAFETY_FENCE_OPEN_32 AT %I* : BOOL;
I_SAFETY_FENCE_LOCK_ON_11 AT %I* : BOOL;
I_SAFETY_FENCE_LOCK_ON_12 AT %I* : BOOL;
I_SAFETY_FENCE_LOCK_ON_13 AT %I* : BOOL;
I_SAFETY_FENCE_LOCK_ON_14 AT %I* : BOOL;
I_SAFETY_FENCE_LOCK_ON_15 AT %I* : BOOL;
I_SAFETY_FENCE_LOCK_ON_16 AT %I* : BOOL;
I_SAFETY_FENCE_LOCK_ON_17 AT %I* : BOOL;
I_SAFETY_FENCE_LOCK_ON_18 AT %I* : BOOL;
I_SAFETY_FENCE_LOCK_ON_21 AT %I* : BOOL;
I_SAFETY_FENCE_LOCK_ON_22 AT %I* : BOOL;
I_SAFETY_FENCE_LOCK_ON_31 AT %I* : BOOL;
I_SAFETY_FENCE_LOCK_ON_32 AT %I* : BOOL;
I_SAFETY_FENCE_LOCK_OFF_11 AT %I* : BOOL;
I_SAFETY_FENCE_LOCK_OFF_12 AT %I* : BOOL;
I_SAFETY_FENCE_LOCK_OFF_13 AT %I* : BOOL;
I_SAFETY_FENCE_LOCK_OFF_14 AT %I* : BOOL;
I_SAFETY_FENCE_LOCK_OFF_15 AT %I* : BOOL;
I_SAFETY_FENCE_LOCK_OFF_16 AT %I* : BOOL;
I_SAFETY_FENCE_LOCK_OFF_17 AT %I* : BOOL;
I_SAFETY_FENCE_LOCK_OFF_18 AT %I* : BOOL;
I_SAFETY_FENCE_LOCK_OFF_21 AT %I* : BOOL;
I_SAFETY_FENCE_LOCK_OFF_22 AT %I* : BOOL;
I_SAFETY_FENCE_LOCK_OFF_31 AT %I* : BOOL;
I_SAFETY_FENCE_LOCK_OFF_32 AT %I* : BOOL;
I_TESTER_ENABLE_11 AT %I* : BOOL;
I_TESTER_ENABLE_12 AT %I* : BOOL;
I_TESTER_ENABLE_13 AT %I* : BOOL;
I_TESTER_ENABLE_14 AT %I* : BOOL;
I_TESTER_ENABLE_15 AT %I* : BOOL;
I_TESTER_ENABLE_16 AT %I* : BOOL;
I_TESTER_ENABLE_17 AT %I* : BOOL;
I_TESTER_ENABLE_18 AT %I* : BOOL;
I_TESTER_ENABLE_21 AT %I* : BOOL;
I_TESTER_ENABLE_22 AT %I* : BOOL;
I_TESTER_ENABLE_31 AT %I* : BOOL;
I_TESTER_ENABLE_32 AT %I* : BOOL;
I_TESTER_DISABLE_11 AT %I* : BOOL;
I_TESTER_DISABLE_12 AT %I* : BOOL;
I_TESTER_DISABLE_13 AT %I* : BOOL;
I_TESTER_DISABLE_14 AT %I* : BOOL;
I_TESTER_DISABLE_15 AT %I* : BOOL;
I_TESTER_DISABLE_16 AT %I* : BOOL;
I_TESTER_DISABLE_17 AT %I* : BOOL;
I_TESTER_DISABLE_18 AT %I* : BOOL;
I_TESTER_DISABLE_21 AT %I* : BOOL;
I_TESTER_DISABLE_22 AT %I* : BOOL;
I_TESTER_DISABLE_31 AT %I* : BOOL;
I_TESTER_DISABLE_32 AT %I* : BOOL;
I_TESTER_EMERGENCY_11 AT %I* : BOOL;
I_TESTER_EMERGENCY_12 AT %I* : BOOL;
I_TESTER_EMERGENCY_13 AT %I* : BOOL;
I_TESTER_EMERGENCY_14 AT %I* : BOOL;
I_TESTER_EMERGENCY_15 AT %I* : BOOL;
I_TESTER_EMERGENCY_16 AT %I* : BOOL;
I_TESTER_EMERGENCY_17 AT %I* : BOOL;
I_TESTER_EMERGENCY_18 AT %I* : BOOL;
I_TESTER_EMERGENCY_21 AT %I* : BOOL;
I_TESTER_EMERGENCY_22 AT %I* : BOOL;
I_TESTER_EMERGENCY_31 AT %I* : BOOL;
I_TESTER_EMERGENCY_32 AT %I* : BOOL;
I_BUFFER_CARRIER_DETECT_1 AT %I* : BOOL;
I_BUFFER_CARRIER_DETECT_2 AT %I* : BOOL;
I_INPUT_CARTESSIAN_HOME AT %I* : BOOL;
I_INPUT_CARTESSIAN_RUNNING AT %I* : BOOL;
I_INPUT_CARTESSIAN_FINISH AT %I* : BOOL;
I_TESTER_READY_11 AT %I* : BOOL;
I_TESTER_READY_12 AT %I* : BOOL;
I_TESTER_READY_13 AT %I* : BOOL;
I_TESTER_READY_14 AT %I* : BOOL;
I_TESTER_READY_15 AT %I* : BOOL;
I_TESTER_READY_16 AT %I* : BOOL;
I_TESTER_READY_17 AT %I* : BOOL;
I_TESTER_READY_18 AT %I* : BOOL;
I_TESTER_READY_21 AT %I* : BOOL;
I_TESTER_READY_22 AT %I* : BOOL;
I_TESTER_READY_31 AT %I* : BOOL;
I_TESTER_READY_32 AT %I* : BOOL;

O_LOADER_CLAMPING_ON_1 AT %Q* : BOOL;
O_LOADER_CLAMPING_ON_2 AT %Q* : BOOL;
O_LOADER_CLAMPING_ON_3 AT %Q* : BOOL;
O_LOADER_CLAMPING_ON_4 AT %Q* : BOOL;
O_LOADER_CLAMPING_OFF_1 AT %Q* : BOOL;
O_LOADER_CLAMPING_OFF_2 AT %Q* : BOOL;
O_LOADER_CLAMPING_OFF_3 AT %Q* : BOOL;
O_LOADER_CLAMPING_OFF_4 AT %Q* : BOOL;
O_C8_GRIPPER_ON AT %Q* : BOOL;
O_C8_GRIPPER_OFF AT %Q* : BOOL;
O_SAFETY_FENCE_LOCK_ON_11 AT %Q* : BOOL;
O_SAFETY_FENCE_LOCK_ON_12 AT %Q* : BOOL;
O_SAFETY_FENCE_LOCK_ON_13 AT %Q* : BOOL;
O_SAFETY_FENCE_LOCK_ON_14 AT %Q* : BOOL;
O_SAFETY_FENCE_LOCK_ON_15 AT %Q* : BOOL;
O_SAFETY_FENCE_LOCK_ON_16 AT %Q* : BOOL;
O_SAFETY_FENCE_LOCK_ON_17 AT %Q* : BOOL;
O_SAFETY_FENCE_LOCK_ON_18 AT %Q* : BOOL;
O_SAFETY_FENCE_LOCK_ON_21 AT %Q* : BOOL;
O_SAFETY_FENCE_LOCK_ON_22 AT %Q* : BOOL;
O_SAFETY_FENCE_LOCK_ON_31 AT %Q* : BOOL;
O_SAFETY_FENCE_LOCK_ON_32 AT %Q* : BOOL;
O_TESTER_TOWER_LAMP_RED_11 AT %Q* : BOOL;
O_TESTER_TOWER_LAMP_RED_12 AT %Q* : BOOL;
O_TESTER_TOWER_LAMP_RED_13 AT %Q* : BOOL;
O_TESTER_TOWER_LAMP_RED_14 AT %Q* : BOOL;
O_TESTER_TOWER_LAMP_RED_15 AT %Q* : BOOL;
O_TESTER_TOWER_LAMP_RED_16 AT %Q* : BOOL;
O_TESTER_TOWER_LAMP_RED_17 AT %Q* : BOOL;
O_TESTER_TOWER_LAMP_RED_18 AT %Q* : BOOL;
O_TESTER_TOWER_LAMP_RED_21 AT %Q* : BOOL;
O_TESTER_TOWER_LAMP_RED_22 AT %Q* : BOOL;
O_TESTER_TOWER_LAMP_RED_31 AT %Q* : BOOL;
O_TESTER_TOWER_LAMP_RED_32 AT %Q* : BOOL;
O_TESTER_TOWER_LAMP_YELLOW_11 AT %Q* : BOOL;
O_TESTER_TOWER_LAMP_YELLOW_12 AT %Q* : BOOL;
O_TESTER_TOWER_LAMP_YELLOW_13 AT %Q* : BOOL;
O_TESTER_TOWER_LAMP_YELLOW_14 AT %Q* : BOOL;
O_TESTER_TOWER_LAMP_YELLOW_15 AT %Q* : BOOL;
O_TESTER_TOWER_LAMP_YELLOW_16 AT %Q* : BOOL;
O_TESTER_TOWER_LAMP_YELLOW_17 AT %Q* : BOOL;
O_TESTER_TOWER_LAMP_YELLOW_18 AT %Q* : BOOL;
O_TESTER_TOWER_LAMP_YELLOW_21 AT %Q* : BOOL;
O_TESTER_TOWER_LAMP_YELLOW_22 AT %Q* : BOOL;
O_TESTER_TOWER_LAMP_YELLOW_31 AT %Q* : BOOL;
O_TESTER_TOWER_LAMP_YELLOW_32 AT %Q* : BOOL;
O_TESTER_TOWER_LAMP_GREEN_11 AT %Q* : BOOL;
O_TESTER_TOWER_LAMP_GREEN_12 AT %Q* : BOOL;
O_TESTER_TOWER_LAMP_GREEN_13 AT %Q* : BOOL;
O_TESTER_TOWER_LAMP_GREEN_14 AT %Q* : BOOL;
O_TESTER_TOWER_LAMP_GREEN_15 AT %Q* : BOOL;
O_TESTER_TOWER_LAMP_GREEN_16 AT %Q* : BOOL;
O_TESTER_TOWER_LAMP_GREEN_17 AT %Q* : BOOL;
O_TESTER_TOWER_LAMP_GREEN_18 AT %Q* : BOOL;
O_TESTER_TOWER_LAMP_GREEN_21 AT %Q* : BOOL;
O_TESTER_TOWER_LAMP_GREEN_22 AT %Q* : BOOL;
O_TESTER_TOWER_LAMP_GREEN_31 AT %Q* : BOOL;
O_TESTER_TOWER_LAMP_GREEN_32 AT %Q* : BOOL;
O_TESTER_CHILLER_ON_11 AT %Q* : BOOL;
O_TESTER_CHILLER_ON_12 AT %Q* : BOOL;
O_TESTER_CHILLER_ON_13 AT %Q* : BOOL;
O_TESTER_CHILLER_ON_14 AT %Q* : BOOL;
O_TESTER_CHILLER_ON_15 AT %Q* : BOOL;
O_TESTER_CHILLER_ON_16 AT %Q* : BOOL;
O_TESTER_CHILLER_ON_17 AT %Q* : BOOL;
O_TESTER_CHILLER_ON_18 AT %Q* : BOOL;
O_TESTER_CHILLER_ON_21 AT %Q* : BOOL;
O_TESTER_CHILLER_ON_22 AT %Q* : BOOL;
O_TESTER_CHILLER_ON_31 AT %Q* : BOOL;
O_TESTER_CHILLER_ON_32 AT %Q* : BOOL;
O_TESTER_CHILLER_OFF_11 AT %Q* : BOOL;
O_TESTER_CHILLER_OFF_12 AT %Q* : BOOL;
O_TESTER_CHILLER_OFF_13 AT %Q* : BOOL;
O_TESTER_CHILLER_OFF_14 AT %Q* : BOOL;
O_TESTER_CHILLER_OFF_15 AT %Q* : BOOL;
O_TESTER_CHILLER_OFF_16 AT %Q* : BOOL;
O_TESTER_CHILLER_OFF_17 AT %Q* : BOOL;
O_TESTER_CHILLER_OFF_18 AT %Q* : BOOL;
O_TESTER_CHILLER_OFF_21 AT %Q* : BOOL;
O_TESTER_CHILLER_OFF_22 AT %Q* : BOOL;
O_TESTER_CHILLER_OFF_31 AT %Q* : BOOL;
O_TESTER_CHILLER_OFF_32 AT %Q* : BOOL;
O_TESTER_POWER_ON_11 AT %Q* : BOOL;
O_TESTER_POWER_ON_12 AT %Q* : BOOL;
O_TESTER_POWER_ON_13 AT %Q* : BOOL;
O_TESTER_POWER_ON_14 AT %Q* : BOOL;
O_TESTER_POWER_ON_15 AT %Q* : BOOL;
O_TESTER_POWER_ON_16 AT %Q* : BOOL;
O_TESTER_POWER_ON_17 AT %Q* : BOOL;
O_TESTER_POWER_ON_18 AT %Q* : BOOL;
O_TESTER_POWER_ON_21 AT %Q* : BOOL;
O_TESTER_POWER_ON_22 AT %Q* : BOOL;
O_TESTER_POWER_ON_31 AT %Q* : BOOL;
O_TESTER_POWER_ON_32 AT %Q* : BOOL;
O_TESTER_PC_SWITCH_ON_11 AT %Q* : BOOL;
O_TESTER_PC_SWITCH_ON_12 AT %Q* : BOOL;
O_TESTER_PC_SWITCH_ON_13 AT %Q* : BOOL;
O_TESTER_PC_SWITCH_ON_14 AT %Q* : BOOL;
O_TESTER_PC_SWITCH_ON_15 AT %Q* : BOOL;
O_TESTER_PC_SWITCH_ON_16 AT %Q* : BOOL;
O_TESTER_PC_SWITCH_ON_17 AT %Q* : BOOL;
O_TESTER_PC_SWITCH_ON_18 AT %Q* : BOOL;
O_TESTER_PC_SWITCH_ON_21 AT %Q* : BOOL;
O_TESTER_PC_SWITCH_ON_22 AT %Q* : BOOL;
O_TESTER_PC_SWITCH_ON_31 AT %Q* : BOOL;
O_TESTER_PC_SWITCH_ON_32 AT %Q* : BOOL;
O_TESTER_START_11 AT %Q* : BOOL;
O_TESTER_START_12 AT %Q* : BOOL;
O_TESTER_START_13 AT %Q* : BOOL;
O_TESTER_START_14 AT %Q* : BOOL;
O_TESTER_START_15 AT %Q* : BOOL;
O_TESTER_START_16 AT %Q* : BOOL;
O_TESTER_START_17 AT %Q* : BOOL;
O_TESTER_START_18 AT %Q* : BOOL;
O_TESTER_START_21 AT %Q* : BOOL;
O_TESTER_START_22 AT %Q* : BOOL;
O_TESTER_START_31 AT %Q* : BOOL;
O_TESTER_START_32 AT %Q* : BOOL;
O_TESTER_STOP_11 AT %Q* : BOOL;
O_TESTER_STOP_12 AT %Q* : BOOL;
O_TESTER_STOP_13 AT %Q* : BOOL;
O_TESTER_STOP_14 AT %Q* : BOOL;
O_TESTER_STOP_15 AT %Q* : BOOL;
O_TESTER_STOP_16 AT %Q* : BOOL;
O_TESTER_STOP_17 AT %Q* : BOOL;
O_TESTER_STOP_18 AT %Q* : BOOL;
O_TESTER_STOP_21 AT %Q* : BOOL;
O_TESTER_STOP_22 AT %Q* : BOOL;
O_TESTER_STOP_31 AT %Q* : BOOL;
O_TESTER_STOP_32 AT %Q* : BOOL;
O_TESTER_EMERGENCY_STOP_11 AT %Q* : BOOL;
O_TESTER_EMERGENCY_STOP_12 AT %Q* : BOOL;
O_TESTER_EMERGENCY_STOP_13 AT %Q* : BOOL;
O_TESTER_EMERGENCY_STOP_14 AT %Q* : BOOL;
O_TESTER_EMERGENCY_STOP_15 AT %Q* : BOOL;
O_TESTER_EMERGENCY_STOP_16 AT %Q* : BOOL;
O_TESTER_EMERGENCY_STOP_17 AT %Q* : BOOL;
O_TESTER_EMERGENCY_STOP_18 AT %Q* : BOOL;
O_TESTER_EMERGENCY_STOP_21 AT %Q* : BOOL;
O_TESTER_EMERGENCY_STOP_22 AT %Q* : BOOL;
O_TESTER_EMERGENCY_STOP_31 AT %Q* : BOOL;
O_TESTER_EMERGENCY_STOP_32 AT %Q* : BOOL;

I_TESTER_JIG_PRESENCE_11 AT %I* : BOOL;
I_TESTER_JIG_PRESENCE_12 AT %I* : BOOL;
I_TESTER_JIG_PRESENCE_13 AT %I* : BOOL;
I_TESTER_JIG_PRESENCE_14 AT %I* : BOOL;
I_TESTER_JIG_PRESENCE_15 AT %I* : BOOL;
I_TESTER_JIG_PRESENCE_16 AT %I* : BOOL;
I_TESTER_JIG_PRESENCE_17 AT %I* : BOOL;
I_TESTER_JIG_PRESENCE_18 AT %I* : BOOL;
I_TESTER_JIG_PRESENCE_21 AT %I* : BOOL;
I_TESTER_JIG_PRESENCE_22 AT %I* : BOOL;
I_TESTER_JIG_PRESENCE_31 AT %I* : BOOL;
I_TESTER_JIG_PRESENCE_32 AT %I* : BOOL;

I_TESTER_BYPASS_TEST_11 AT %I* : BOOL;
I_TESTER_BYPASS_TEST_12 AT %I* : BOOL;
I_TESTER_BYPASS_TEST_13 AT %I* : BOOL;
I_TESTER_BYPASS_TEST_14 AT %I* : BOOL;
I_TESTER_BYPASS_TEST_15 AT %I* : BOOL;
I_TESTER_BYPASS_TEST_16 AT %I* : BOOL;
I_TESTER_BYPASS_TEST_17 AT %I* : BOOL;
I_TESTER_BYPASS_TEST_18 AT %I* : BOOL;
I_TESTER_BYPASS_TEST_21 AT %I* : BOOL;
I_TESTER_BYPASS_TEST_22 AT %I* : BOOL;
I_TESTER_BYPASS_TEST_31 AT %I* : BOOL;
I_TESTER_BYPASS_TEST_32 AT %I* : BOOL;

END_VAR

// ---- GVLs/POWER_CONTROL.TcGVL
{attribute 'qualified_only'}
VAR_GLOBAL
O_PWR_CTRL_ROBOT_G6 AT %Q* : BOOL;
O_PWR_CTRL_ROBOT_RS4_1 AT %Q* : BOOL;
O_PWR_CTRL_ROBOT_RS4_2 AT %Q* : BOOL;
O_PWR_CTRL_ROBOT_C8 AT %Q* : BOOL;
O_PWR_CTRL_STEPDOWN AT %Q* : BOOL;
O_PWR_CTRL_INDEXING_1 AT %Q* : BOOL;//O_PWR_CONTROL_24V_INDEXING_ROTARY AT %Q* : BOOL;
O_PWR_CTRL_INDEXING_2 AT %Q* : BOOL;//O_PWR_CONTROL_24V_STRAIGHTENER_GRIPPER_EXT AT %Q* : BOOL;
O_PWR_CTRL_PC_1 AT %Q* : BOOL;

O_G6_HOME AT %Q* : BOOL;
O_RS4_HOME_1 AT %Q* : BOOL;
O_RS4_HOME_2 AT %Q* : BOOL;
O_C8_HOME_1 AT %Q* : BOOL;
O_INDEXING_HOME_1 AT %Q* : BOOL;
O_INDEXING_HOME_2 AT %Q* : BOOL;

END_VAR

// ---- GVLs/SORTER_RS4_VAR.TcGVL
{attribute 'qualified_only'}
VAR_GLOBAL

SORTER_RS4_INPUT AT %IB64 : BYTE;  
SORTER_RS4_INPUT_1 AT %IB65 : BYTE; 
SORTER_RS4_INPUT_2 AT %IB66 : BYTE;  
SORTER_RS4_INPUT_3 AT %IB67 : BYTE; 
SORTER_RS4_INPUT_4 AT %IB68 : BYTE; 
SORTER_RS4_INPUT_5 AT %IB69 : BYTE; 
SORTER_RS4_INPUT_6 AT %IB70 : BYTE; 

SORTER_RS4_OUTPUT AT %QB64 : BYTE; 
SORTER_RS4_OUTPUT_1 AT %QB65 : BYTE; 
SORTER_RS4_POS_TAKEUP_1 AT %QB66 : BYTE:=1; 
SORTER_RS4_POS_TAKEUP_2 AT %QB67 : BYTE:=2;
SORTER_RS4_POS_TAKEUP_3 AT %QB68 : BYTE:=3; 
SORTER_RS4_POS_TAKEUP_4 AT %QB69 : BYTE:=4;
SORTER_RS4_POS_PLACING_1 AT %QB70 : BYTE:=1; 
SORTER_RS4_POS_PLACING_2 AT %QB71 : BYTE:=5;
SORTER_RS4_POS_PLACING_3 AT %QB72 : BYTE:=9; 
SORTER_RS4_POS_PLACING_4 AT %QB73 : BYTE:=9; 
I_SORTER_RS4_READY_TAKEUP  AT %IX67.2 :BOOL;//CYCLE RUNNING INDICATOR
I_SORTER_RS4_START_TAKEUP  AT %IX67.3 :BOOL;
I_SORTER_RS4_READY_PLACING  AT %IX67.4 :BOOL;
I_SORTER_RS4_START_PLACING  AT %IX67.5 :BOOL;
O_SORTER_RS4_CONTINUE AT %QX64.6  : BOOL;
I_SORTER_RS4_HANG :BOOL;
I_SORTER_RS4_END_CARRIER :BOOL:=true;
I_SORTER_RS4_ENABLE :BOOL; 
I_SORTER_RS4_DISABLE :BOOL;

SORTER_RS4_OUTPUT_10 AT %QB74 : BYTE;

I_SORTER_RS4_READY  AT %IX64.0 :BOOL;
I_SORTER_RS4_RUNNING  AT %IX64.1 :BOOL;
I_SORTER_RS4_PAUSED  AT %IX64.2 :BOOL;
I_SORTER_RS4_ERROR  AT %IX64.3 :BOOL;
I_SORTER_RS4_ESTOPON  AT %IX64.4 :BOOL;
I_SORTER_RS46_SAFEGUARDON  AT %IX64.5 :BOOL;
I_SORTER_RS4_SERROR  AT %IX64.6 :BOOL;
I_SORTER_RS4_WARNING  AT %IX64.7 :BOOL;

I_SORTER_RS4_MOTORON  AT %IX65.0 :BOOL;
I_SORTER_RS4_ATHOME  AT %IX65.1 :BOOL;
I_SORTER_RS4_AUTOMODE  AT %IX65.5 :BOOL;

IX_SORTER_RS4_GRIPPER_1 AT %IX66.0 : BOOL;
IX_SORTER_RS4_GRIPPER_2 AT %IX66.1 : BOOL;
IX_SORTER_RS4_GRIPPER_3 AT %IX66.2 : BOOL;
IX_SORTER_RS4_GRIPPER_4 AT %IX66.3 : BOOL;

IX_SORTER_RS4_GRIPPER_EXT_1 AT %IX66.4 : BOOL;
IX_SORTER_RS4_GRIPPER_EXT_2 AT %IX66.5 : BOOL;
IX_SORTER_RS4_GRIPPER_EXT_3 AT %IX66.6 : BOOL;
IX_SORTER_RS4_GRIPPER_EXT_4 AT %IX66.7 : BOOL;

I_SORTER_RS4_END_CYCLE  AT %IX67.0 :BOOL;
//I_SORTER_RS4_END_CARRIER  AT %IX69.1 :BOOL;
	
	O_SORTER_RS4_START AT %QX64.0  : BOOL;	
	O_SORTER_RS4_SELECT_FUKUDA_A AT %QX64.1  : BOOL;
	O_SORTER_RS4_SELECT_FUKUDA_B AT %QX64.2  : BOOL;
	O_SORTER_RS4_STOP AT %QX64.4  : BOOL;
	O_SORTER_RS4_PAUSE AT %QX64.5  : BOOL;
	O_SORTER_RS4_RESET AT %QX64.7  : BOOL;	
	
	O_SORTER_RS4_SETMOTORON AT %QX65.0  : BOOL;
	O_SORTER_RS4_SETMOTOROFF AT %QX65.1  : BOOL;
	O_SORTER_RS4_HOME AT %QX65.2  : BOOL;

I_SORTER_RS4_GRIPPER_CLOSE_1 AT %I* : BOOL;
I_SORTER_RS4_GRIPPER_CLOSE_2 AT %I* : BOOL;
I_SORTER_RS4_GRIPPER_CLOSE_3 AT %I* : BOOL;
I_SORTER_RS4_GRIPPER_CLOSE_4 AT %I* : BOOL;
I_SORTER_RS4_GRIPPER_OPEN_1 AT %I* : BOOL;
I_SORTER_RS4_GRIPPER_OPEN_2 AT %I* : BOOL;
I_SORTER_RS4_GRIPPER_OPEN_3 AT %I* : BOOL;
I_SORTER_RS4_GRIPPER_OPEN_4 AT %I* : BOOL;
I_SORTER_RS4_GRIPPER_EXT_DOWN_1 AT %I* : BOOL;
I_SORTER_RS4_GRIPPER_EXT_DOWN_2 AT %I* : BOOL;
I_SORTER_RS4_GRIPPER_EXT_DOWN_3 AT %I* : BOOL;
I_SORTER_RS4_GRIPPER_EXT_DOWN_4 AT %I* : BOOL;
I_SORTER_RS4_GRIPPER_EXT_UP_1 AT %I* : BOOL;
I_SORTER_RS4_GRIPPER_EXT_UP_2 AT %I* : BOOL;
I_SORTER_RS4_GRIPPER_EXT_UP_3 AT %I* : BOOL;
I_SORTER_RS4_GRIPPER_EXT_UP_4 AT %I* : BOOL;

O_SORTER_RS4_GRIPPER_CLOSE_1 AT %Q* : BOOL;
O_SORTER_RS4_GRIPPER_CLOSE_2 AT %Q* : BOOL;
O_SORTER_RS4_GRIPPER_CLOSE_3 AT %Q* : BOOL;
O_SORTER_RS4_GRIPPER_CLOSE_4 AT %Q* : BOOL;
O_SORTER_RS4_GRIPPER_OPEN_1 AT %Q* : BOOL;
O_SORTER_RS4_GRIPPER_OPEN_2 AT %Q* : BOOL;
O_SORTER_RS4_GRIPPER_OPEN_3 AT %Q* : BOOL;
O_SORTER_RS4_GRIPPER_OPEN_4 AT %Q* : BOOL;
O_SORTER_RS4_GRIPPER_EXT_DOWN_1 AT %Q* : BOOL;
O_SORTER_RS4_GRIPPER_EXT_DOWN_2 AT %Q* : BOOL;
O_SORTER_RS4_GRIPPER_EXT_DOWN_3 AT %Q* : BOOL;
O_SORTER_RS4_GRIPPER_EXT_DOWN_4 AT %Q* : BOOL;
O_SORTER_RS4_GRIPPER_EXT_UP_1 AT %Q* : BOOL;
O_SORTER_RS4_GRIPPER_EXT_UP_2 AT %Q* : BOOL;
O_SORTER_RS4_GRIPPER_EXT_UP_3 AT %Q* : BOOL;
O_SORTER_RS4_GRIPPER_EXT_UP_4 AT %Q* : BOOL;

IX_SORTER_RS4_HOME AT %I* : BOOL;
IX_SORTER_RS4_RUNNING AT %I* : BOOL;
IX_SORTER_RS4_PICKUP_1 AT %I* : BOOL;
IX_SORTER_RS4_PICKUP_2 AT %I* : BOOL;
IX_SORTER_RS4_PICKUP_3 AT %I* : BOOL;
IX_SORTER_RS4_PICKUP_4 AT %I* : BOOL;
IX_SORTER_RS4_PLACING_1 AT %I* : BOOL;
IX_SORTER_RS4_PLACING_2 AT %I* : BOOL;
IX_SORTER_RS4_PLACING_3 AT %I* : BOOL;
IX_SORTER_RS4_PLACING_4 AT %I* : BOOL;

IX_SORTER_RS4_FINISH AT %I* : BOOL;
READY_INDEXING :BOOL;
END_VAR

// ---- GVLs/SORTER_VAR.TcGVL
{attribute 'qualified_only'}
VAR_GLOBAL
I_LOTBOX_CLAMP_ON_1 AT %I* : BOOL;
I_LOTBOX_CLAMP_ON_2 AT %I* : BOOL;
I_LOTBOX_CLAMP_ON_3 AT %I* : BOOL;
I_LOTBOX_CLAMP_ON_4 AT %I* : BOOL;
I_LOTBOX_CLAMP_OFF_1 AT %I* : BOOL;
I_LOTBOX_CLAMP_OFF_2 AT %I* : BOOL;
I_LOTBOX_CLAMP_OFF_3 AT %I* : BOOL;
I_LOTBOX_CLAMP_OFF_4 AT %I* : BOOL;
	
I_LOTBOX_DETECT_1 AT %I* : BOOL;//LOTBOX_LASER1_DETECT
I_LOTBOX_DETECT_2 AT %I* : BOOL;//LOTBOX_LASER2_DETECT
I_LOTBOX_DETECT_3 AT %I* : BOOL;//LOTBOX_LASER3_DETECT
I_LOTBOX_DETECT_4 AT %I* : BOOL;//LOTBOX_LASER4_DETECT

I_VACUUM_ON AT %I* : BOOL;
I_VACUUM_OFF AT %I* : BOOL;

I_RETURN_DONE_A: BOOL;
I_RETURN_DONE_B: BOOL;
I_RETURN_DONE_NG: BOOL;
I_LOADING_DONE_A: BOOL;
I_LOADING_DONE_B: BOOL;
I_LOADING_DONE_NG : BOOL; 
I_LASER_ONDUTY_A:BOOL;
I_LASER_ONDUTY_B:BOOL;
I_LASER_ONDUTY_NG:BOOL;
I_LASER_SOCKET : T_JIG_SOCKET; 
I_CURRENT_TRANSACTION : T_CURRENT_TRANSACTION ;
I_LASER_TRANSFER_AT_FRONT_A AT %I* : BOOL;
I_LASER_TRANSFER_AT_BACK_A AT %I* : BOOL;
I_LASER_TRANSFER_AT_FRONT_B AT %I* : BOOL;
I_LASER_TRANSFER_AT_BACK_B AT %I* : BOOL;
I_NG_TRANSFER_AT_FRONT_B AT %I* : BOOL;
I_NG_TRANSFER_AT_BACK_B AT %I* : BOOL;
I_LASER_TRANSFER_A_PICK_DONE : BOOL;
I_LASER_TRANSFER_B_PICK_DONE : BOOL;
I_LASER_TRANSFER_AT_A : BOOL;
I_LASER_TRANSFER_AT_B : BOOL;
I_FUKUDA_TRANSFER_A_PICKING:BOOL;
I_LOTEND:BOOL;
I_LASER_TRANSFER_A_PICKING:BYTE;

//I_LOTEND :BOOL :=FALSE;
I_CARTESSIAN_GRIPPER_ON AT %I* : BOOL;
I_CARTESSIAN_GRIPPER_OFF AT %I* : BOOL;
I_FUNCTION_NAME :STRING [255];
I_CASE : INT:=0;
I_NG_CASE : INT :=100;
I_LASER_RUNNING:BOOL :=FALSE;

O_LOTBOX_CLAMP_ON_1 AT %Q* : BOOL;
O_LOTBOX_CLAMP_ON_2 AT %Q* : BOOL;
O_LOTBOX_CLAMP_ON_3 AT %Q* : BOOL;
O_LOTBOX_CLAMP_ON_4 AT %Q* : BOOL;
O_LOTBOX_CLAMP_OFF_1 AT %Q* : BOOL;
O_LOTBOX_CLAMP_OFF_2 AT %Q* : BOOL;
O_LOTBOX_CLAMP_OFF_3 AT %Q* : BOOL;
O_LOTBOX_CLAMP_OFF_4 AT %Q* : BOOL;

O_VACUUM_ON AT %Q* : BOOL;
O_VACUUM_OFF AT %Q* : BOOL;
O_CARTESSIAN_GRIPPER_ON AT %Q* : BOOL;
O_CARTESSIAN_GRIPPER_OFF AT %Q* : BOOL;
O_TOWER_LAMP_RED AT %Q* : BOOL;
O_TOWER_LAMP_YELLOW AT %Q* : BOOL;
O_TOWER_LAMP_GREEN AT %Q* : BOOL;
O_TOWER_LAMP_BUZZER AT %Q* : BOOL;
O_WARNING_LIGHT AT %Q* : BOOL;
O_LOT_BOX_INDICATOR_1  AT %Q* : BOOL;
O_LOT_BOX_INDICATOR_2 AT %Q* : BOOL;
O_LOT_BOX_INDICATOR_3 AT %Q* : BOOL;
O_LOT_BOX_INDICATOR_4 AT %Q* : BOOL;

AXIS_COMPLETE: BOOL;
JIG_LASER_PRESENCE: BOOL;
LOTBOX_READY_1: BOOL;

DataWordInput1 AT %IB232 : ARRAY [0..15] OF WORD; 
DataWordInput2 AT %IB264 : ARRAY [16..31] OF WORD;
DataWordInput3 AT %IB296 : ARRAY [32..47] OF WORD; 
DataWordInput4 AT %IB328 : ARRAY [48..56] OF WORD; 
DataWordOutput1 AT %QB232 : ARRAY [0..15] OF WORD; 
DataWordOutput2 AT %QB264 : ARRAY [16..31] OF WORD; 
DataWordOutput3 AT %QB296 : ARRAY [32..47] OF WORD; 
DataWordOutput4 AT %QB328 : ARRAY [48..56] OF WORD; 

I_NG_BUFFER_ON AT %I* : BOOL;
I_NG_BUFFER_OFF AT %I* : BOOL;
I_NG_BOX_DETECT_1 AT %I* : BOOL;
I_NG_BOX_DETECT_2 AT %I* : BOOL;
I_NG_BOX_DETECT_3 AT %I* : BOOL;
I_NG_BOX_DETECT_4 AT %I* : BOOL;
I_NG_HOME :BOOL;
I_NG_TRANSFER_AT_BACK AT %I* : BOOL;
I_NG_TRANSFER_AT_FRONT AT %I* : BOOL;

O_NG_DATA_OUTPUT1 AT %Q* : BOOL;
O_NG_DATA_OUTPUT2 AT %Q* : BOOL;
O_NG_DATA_OUTPUT3 AT %Q* : BOOL;
O_NG_DATA_OUTPUT4 AT %Q* : BOOL;
O_NG_BUFFER_ON AT %Q* : BOOL;
O_NG_BUFFER_OFF AT %Q* : BOOL;
O_NG_HOMING :BOOL;
O_NG_BOX_INDICATOR_1 AT %Q* : BOOL;
O_NG_BOX_INDICATOR_2 AT %Q* : BOOL;
O_NG_BOX_INDICATOR_3 AT %Q* : BOOL;
O_NG_BOX_INDICATOR_4 AT %Q* : BOOL;
O_NG_DATA_STOP AT %Q* : BOOL;
O_NG_DATA_RESET AT %Q* : BOOL;
RETURN_NG_IDX:BYTE;
LOAD_NG_IDX:BYTE;
//I_RETURN_DONE_A: BOOL;
//I_RETURN_DONE_B: BOOL;
//I_LOADING_DONE_A: BOOL;
//I_LOADING_DONE_B: BOOL;
I_RETURN_ALARM: INT;
I_RETURN_FAILED: BOOL;
ACTIVE_ID: INT :=1;	
ACTIVE_PROGRAM: INT ;
ACTIVE_PROGRAM_CHANGE:BOOL;
	
I_LASER_HOME : BOOL;
O_LASER_HOME : BOOL;

STRAIGHTEN_START: BOOL;
STRAIGHTEN_PROCESS: BOOL;
STRAIGHTEN_DONE: BOOL;

LASER_HOME: BOOL;

O_STOPPER_TRANSFER_A AT %Q* : BOOL;
O_STOPPER_TRANSFER_B AT %Q* : BOOL;
I_STOPPER_TRANSFER_ON_A AT %Q* : BOOL;
I_STOPPER_TRANSFER_OFF_A AT %Q* : BOOL;
I_STOPPER_TRANSFER_ON_B AT %Q* : BOOL;
I_STOPPER_TRANSFER_OFF_B AT %Q* : BOOL;
O_RESET_CARTESSIAN AT %Q* : BOOL;

TRANSPORT_IDX: BYTE;
STATION_LOAD_IDX: BYTE;
STATION_RETURN_IDX: BYTE;
JIG_LOAD_IDX: BYTE;
JIG_RETURN_IDX: BYTE;

END_VAR

// ---- GVLs/TESTER_C8_VAR.TcGVL
{attribute 'qualified_only'}
VAR_GLOBAL
C8_MACHINE_POSITION : T_MACHINE_POSITION;
C8_MACHINE_POSITION_TAKE : T_MACHINE_POSITION;

I_C8_JIG_PRESENCE AT %IX204.7 : BOOL;
O_G6_FINISH_SCANBARCODE AT %QX202.0 : BOOL;

C8_STATE_1 	AT %IB200 : BYTE;
C8_STATE_2 	AT %IB201 : BYTE;
C8_ERROR_1 	AT %IB202 : BYTE;
C8_ERROR_2 	AT %IB203 : BYTE;
C8_INPUT_1 	AT %IB204 : BYTE;

C8_CONTROL_1 AT %QB200 : BYTE;
C8_CONTROL_2 AT %QB201 : BYTE;
C8_CONTROL_3 AT %QB202 : BYTE;
C8_INDEX_POSITION AT %QB203 : BYTE;
C8_MOVEMENT_SOURCE AT %QB204 : BYTE ;
C8_MOVEMENT_DESTINATION AT %QB205 : BYTE ;

I_C8_READY  AT %IX200.0 :BOOL;
I_C8_RUNNING  AT %IX200.1 :BOOL;
I_C8_PAUSED  AT %IX200.2 :BOOL;
I_C8_ERROR  AT %IX200.3 :BOOL;
I_C8_ESTOPON  AT %IX200.4 :BOOL;
I_C8_SAFEGUARDON  AT %IX200.5 :BOOL;
I_C8_SERROR  AT %IX200.6 :BOOL;
I_C8_WARNING  AT %IX200.7 :BOOL;

I_C8_MOTORON  AT %IX201.0 :BOOL;
I_C8_ATHOME  AT %IX201.1 :BOOL;
I_C8_AUTOMODE  AT %IX201.5 :BOOL;
I_C8_TEACHMODE  AT %IX201.6 :BOOL;

I_C8_GRIPPER AT %IX204.0 : BOOL;
I_C8_FREE AT %IX204.1 : BOOL;
I_C8_READY_SCAN AT %IX204.2 : BOOL;
I_C8_ROTATE_INDEXING_2 AT %IX204.3 : BOOL;
I_C8_MCAL_REQUEST AT %IX204.4 : BOOL;
O_C8_GRIPPER_CLOSE AT %Q*: BOOL;
O_C8_GRIPPER_OPEN AT %Q* : BOOL;
	
	O_G6_START AT %QX200.0  : BOOL;	
	O_G6_SELPROG1 AT %QX200.1  : BOOL;
	O_G6_SELPROG2 AT %QX200.2  : BOOL;
	O_G6_SELPROG4 AT %QX200.3  : BOOL;
	O_G6_STOP AT %QX200.4  : BOOL;
	O_G6_PAUSE AT %QX200.5  : BOOL;
	O_G6_CONTINUE AT %QX200.6  : BOOL;
	O_G6_RESET AT %QX200.7  : BOOL;	
	
	O_G6_SETMOTORON AT %QX201.0  : BOOL;
	O_G6_SETMOTOROFF AT %QX201.1  : BOOL;
	O_G6_HOME AT %QX201.2  : BOOL;
	O_G6_SHUTDOWN AT %QX201.3  : BOOL;
	O_G6_MCAL AT %QX201.4  : BOOL;
	O_G6_SELROBOT AT %QX201.5  : BOOL;
	O_G6_SELROBOT_1 AT %QX201.6  : BOOL;
	O_G6_SELROBOT_2 AT %QX201.7  : BOOL;
	
	

O_C8_ENABLE :BOOL :=TRUE;
C8_PUTON: BOOL;
C8_TAKING: BOOL;
C8_TRANSFER: BOOL;
C8_ONDUTY:BOOL;
C8_START_MOVING :BOOL;

READY_INDEXING :BOOL;
END_VAR

// ---- POUs/FUKUDA/FUKUDA_MOVE.TcPOU
PROGRAM FUKUDA_MOVE
//FUNCTION FUKUDA_MOVE : BOOL
VAR_INPUT
	STEP_DATA_1: BYTE;
	STEP_DATA_2: BYTE;
	STEP_DATA_3: BYTE;
	STEP_DATA_4: BYTE;
	STEP_DATA_5: BYTE;
	FUKUDA_HOME: INT;
END_VAR

VAR
	
	(*
	DataWordInput1 AT %IB100 : ARRAY [0..15] OF WORD; 
	DataWordInput2 AT %IB132 : ARRAY [16..31] OF WORD; 
	DataWordInput3 AT %IB164 : ARRAY [32..47] OF WORD; 
	DataWordInput4 AT %IB196 : ARRAY [48..56] OF WORD; 
	DataWordOutput1 AT %QB100 : ARRAY [0..15] OF WORD; 
	DataWordOutput2 AT %QB132 : ARRAY [16..31] OF WORD; 
	DataWordOutput3 AT %QB164 : ARRAY [32..47] OF WORD; 
	DataWordOutput4 AT %QB196 : ARRAY [48..56] OF WORD; 
	*)
	Gateway_Q0_MODE_COMMAND_0 AT %QX100.0 : BOOL ;
	Gateway_Q0_MODE_COMMAND_1 AT %QX100.1 : BOOL ;
	Gateway_Q0_RESET AT %QX100.4 : BOOL;
	Gateway_Q0_RESTART AT %QX100.5 : BOOL;
	Gateway_Q0_STOP AT %QX100.7 : BOOL;
	Gateway_Q1_0 AT %QX101.0 : BOOL;
	Gateway_Q1_1 AT %QX101.1 : BOOL;
	Gateway_Q1_2 AT %QX101.2 : BOOL;
	Gateway_Q1_3 AT %QX101.3 : BOOL;
	Gateway_Q1_4 AT %QX101.4 : BOOL;
	Gateway_Gateway_Unit_2_Status AT %QB102 : BYTE;
	Gateway_Q3_0 AT %QX103.0 : BOOL;
	Gateway_Q3_1 AT %QX103.1 : BOOL;
	Gateway_Q3_2 AT %QX103.2 : BOOL;
	Gateway_Q3_3 AT %QX103.3 : BOOL;	
	

	ID1_StepData AT %QB114 : BYTE;
	ID1_Hold AT %QX115.0 : BOOL;
	ID1_SVON AT %QX115.1 : BOOL;
	ID1_Drive AT %QX115.2 : BOOL;
	ID1_Reset AT %QX115.3 : BOOL;
	ID1_Setup AT %QX115.4 : BOOL;
	

	ID2_StepData AT %QB134 : BYTE;
	ID2_Hold AT %QX135.0 : BOOL;
	ID2_SVON AT %QX135.1 : BOOL;
	ID2_Drive AT %QX135.2 : BOOL;
	ID2_Reset AT %QX135.3 : BOOL;
	ID2_Setup AT %QX135.4 : BOOL;


	ID3_StepData AT %QB154 : BYTE;
	ID3_Hold AT %QX155.0 : BOOL;
	ID3_SVON AT %QX155.1 : BOOL;
	ID3_Drive AT %QX155.2 : BOOL;
	ID3_Reset AT %QX155.3 : BOOL;
	ID3_Setup AT %QX155.4 : BOOL;
	
	
	ID4_StepData AT %QB174 : BYTE;
	ID4_Hold AT %QX175.0 : BOOL;
	ID4_SVON AT %QX175.1 : BOOL;
	ID4_Drive AT %QX175.2 : BOOL;
	ID4_Reset AT %QX175.3 : BOOL;
	ID4_Setup AT %QX175.4 : BOOL;
	

	ID5_StepData AT %QB194 : BYTE;
	ID5_Hold AT %QX195.0 : BOOL;
	ID5_SVON AT %QX195.1 : BOOL;
	ID5_Drive AT %QX195.2 : BOOL;
	ID5_Reset AT %QX195.3 : BOOL;
	ID5_Setup AT %QX195.4 : BOOL;
	
	byte0 : BYTE;
	byte1 : BYTE;
	byte2 : BYTE;
	byte3 : BYTE;
	
	bit14_0 : BOOL;
	bit14_1 : BOOL;
	bit14_2 : BOOL;
	bit14_3 : BOOL;
	bit14_4 : BOOL;
	bit14_5 : BOOL;
	
	bit15_0 : BOOL;
	bit15_1 : BOOL;
	bit15_2 : BOOL;
	bit15_3 : BOOL;
	bit15_4 : BOOL; 
	
	bit34_0 : BOOL;
	bit34_1 : BOOL;
	bit34_2 : BOOL;
	bit34_3 : BOOL;
	bit34_4 : BOOL;
	bit34_5 : BOOL;
	
	bit35_0 : BOOL;
	bit35_1 : BOOL;
	bit35_2 : BOOL;
	bit35_3 : BOOL;
	bit35_4 : BOOL; 
	
	bit54_0 : BOOL;
	bit54_1 : BOOL;
	bit54_2 : BOOL;
	bit54_3 : BOOL;
	bit54_4 : BOOL;
	bit54_5 : BOOL;
	
	bit55_0 : BOOL;
	bit55_1 : BOOL;
	bit55_2 : BOOL;
	bit55_3 : BOOL;
	bit55_4 : BOOL; 
	
	bit74_0 : BOOL;
	bit74_1 : BOOL;
	bit74_2 : BOOL;
	bit74_3 : BOOL;
	bit74_4 : BOOL;
	bit74_5 : BOOL;
	
	bit75_0 : BOOL;
	bit75_1 : BOOL;
	bit75_2 : BOOL;
	bit75_3 : BOOL;
	bit75_4 : BOOL; 
	
	bit94_0 : BOOL;
	bit94_1 : BOOL;
	bit94_2 : BOOL;
	bit94_3 : BOOL;
	bit94_4 : BOOL;
	bit94_5 : BOOL;
	
	bit95_0 : BOOL;
	bit95_1 : BOOL;
	bit95_2 : BOOL;
	bit95_3 : BOOL;
	bit95_4 : BOOL; 	
	
	ID1_I0_MODE_COMMAND_0 AT %IX100.0 : BOOL :=0;
	ID1_I0_MODE_COMMAND_1 AT %IX100.1 : BOOL:=0;
	ID1_I0_READY AT %IX100.4 : BOOL;
	ID1_I0_ALARM AT %IX100.5 : BOOL;
	ID1_I0_INITIAL AT %IX100.6 : BOOL;
	ID1_I0_COMMUNICATING AT %IX100.7 : BOOL;
	ID1_I1_0 AT %IX101.0 : BOOL;
	ID1_I1_1 AT %IX101.1 : BOOL;
	ID1_I1_2 AT %IX101.2 : BOOL;
	ID1_I1_3 AT %IX101.3 : BOOL;
	ID1_I1_4 AT %IX101.4 : BOOL;
	ID1_I2_0 AT %IX102.0 : BOOL;
	ID1_I2_1 AT %IX102.1 : BOOL;
	ID1_I2_2 AT %IX102.2 : BOOL;
	ID1_I2_3 AT %IX102.3 : BOOL;
	ID1_I2_4 AT %IX102.4 : BOOL;

	ID1_I3_0 AT %IX103.0 : BOOL;
	ID1_I3_1 AT %IX103.1 : BOOL;
	
	ID1_I32_0 AT %IX132.0 : BOOL;
	ID1_I32_1 AT %IX132.1 : BOOL;
	ID1_I33_0 AT %IX133.0 : BOOL;
	ID1_I33_1 AT %IX133.1 : BOOL;
(*-----------------------------------------------------------*)

	iTest15: SINT;
	iTest16: SINT;
	
	bTest1 : BOOL;
	bTest2 : BOOL;
	bTest3 : BOOL;
	bTest4 : BOOL;
	bTest5 : BOOL;
	bTest6 : BOOL;
	bTest7 : BOOL;
	bTest8 : BOOL;
	bTest9 : BOOL;
	bTest10 : BOOL;
	bTest11 : BOOL;
	bTest12 : BOOL;
	bTest13 : BOOL;
	bTest14 : BOOL;
	
	StepData1 : BYTE;
	StepData2 : BYTE;
	StepData3 : BYTE;
	StepData4 : BYTE;
	StepData5 : BYTE;
	
	star :BOOL;
	hom : BOOL;

	reset: BOOL;
	
	ID1_ALARM AT%IX115.7 : BOOL;
	ID2_ALARM AT%IX135.7 : BOOL;
	ID3_ALARM AT%IX155.7 : BOOL;
	ID4_ALARM AT%IX175.7 : BOOL;
	ID5_ALARM AT%IX195.7 : BOOL;
	
	ID1_SVRE AT%IX115.1 : BOOL;
	ID2_SVRE AT%IX135.1 : BOOL;
	ID3_SVRE AT%IX155.1 : BOOL;
	ID4_SVRE AT%IX175.1 : BOOL;
	ID5_SVRE AT%IX195.1 : BOOL;
	
	ID1_INP AT%IX115.3 : BOOL;
	ID2_INP AT%IX135.3 : BOOL;
	ID3_INP AT%IX155.3 : BOOL;
	ID4_INP AT%IX175.3 : BOOL;
	ID5_INP AT%IX195.3 : BOOL;
	
	PROSES: STRING;
	STAGE: INT;
	
	PROCESS: INT;
	START_PROCESS: BOOL;
	STEP_DATAS: INT;
	PROCESS_DELAY: TIME :=T#300MS;
	FUKUDA_RUNNING: BOOL :=FALSE;
	ACTIVE_STEPDATA : BYTE;
	//ACTIVE_ID: INT :=1;
	TMR1: TON;
	TMR2: TON;
	TMR3: TON;
	TMR4: TON;
	TMR5: TON;
	TMR6: TON;
	TMR10: Ton;
	TMR11: TON;
	TMR12: TON;
	TMR13: TON;
	TMR14: TON;
	TMR20: TON;
	TMR21: TON;
	TMR22: TON;
	TMR23: TON;
	TMR30: TON;
	TMR31: TON;
	TMR32: TON;
	TMR33: TON;
	TMR40: TON;
	TMR41: TON;
	TMR42: TON;
	TMR43: TON;
	TMR50: TON;
	TMR51: TON;
	TMR52: TON;
	TMR53: TON;
	
	
	TMR101: TON;
	TMR102: TON;
	TMR103: TON;
	TMR104: TON;
	TMR105: TON;
	TMR106: TON;
	ID5: INT;
	TMR7: Ton;
	TMR_RES_CARTSN: TOF;
	TMR_ACTIVATE_RESET: TON;
	ID3_READY: BOOL;
	ID2_READY: BOOL;
	ID1_READY: BOOL;
	ID4_READY: BOOL;
	ID5_READY: BOOL;
END_VAR


PROCESS_DELAY:= T#400MS;
IF 	INPUT_VAR.ACTIVE_ID >=0 THEN
STEP_DATA_1:=STEP_DATA_1+1;

IF STEP_DATA_2>=5 THEN
	STEP_DATA_2:=STEP_DATA_2+1;
END_IF

STEP_DATA_3:=STEP_DATA_3+1;	
END_IF


IF NOT INPUT_VAR.FUKUDA_HOME THEN //fukuda_running THEN
	IF  ID1_SVRE AND ID2_SVRE  AND  ID3_SVRE AND  ID4_SVRE AND  ID5_SVRE THEN
		TMR1(IN:=TRUE,PT:=T#0.5S);
		TMR4(IN:=TRUE,PT:=T#3S);
		TMR5(IN:=TRUE,PT:=T#3.5S);
		TMR6(IN:=TRUE,PT:=T#25S);

		IF ID2_SVRE THEN
			ID2_SETUP :=TRUE;
			IF ID2_INP THEN
				ID2_READY:=TRUE;
				IF ID3_SVRE THEN
					ID3_SETUP :=TRUE;
					IF ID3_INP THEN
						ID3_READY:=TRUE;
						IF ID1_SVRE THEN
							ID1_SETUP :=TRUE;
							IF ID1_INP THEN
								ID1_READY:=TRUE;
							END_IF
						ELSE
							ID1_SVON :=TRUE;	
						END_IF
					END_IF
				ELSE
					ID3_SVON :=TRUE;	
				END_IF
			END_IF
		ELSE
			ID2_SVON :=TRUE;	
		END_IF
	
	IF ID1_INP THEN		
		CASE INPUT_VAR.I_CURRENT_TRANSACTION.TRANSPORT_INDEX OF
		1:
			TMR2(IN:=TRUE,PT:=T#1S);
			IF ID4_SVRE THEN
				ID4_SETUP :=TRUE;
				IF ID4_INP THEN
					ID4_READY:=TRUE;
				END_IF
			ELSE
				ID4_SVON :=TRUE;	
			END_IF
		2:
			TMR3(IN:=TRUE,PT:=T#1.5S);
			IF ID5_SVRE THEN
				ID5_SETUP :=TRUE;
				IF ID5_INP THEN
					ID5_READY:=TRUE;
				END_IF
			ELSE
				ID5_SVON :=TRUE;	
			END_IF
		END_CASE
	END_IF
	//IF TMR6.Q THEN
	IF ID1_INP AND ID2_INP AND ID3_INP AND (ID4_INP OR ID5_INP) THEN
		ID1_SETUP :=FALSE;
		ID2_SETUP :=FALSE;
		ID3_SETUP :=FALSE;
		ID4_SETUP :=FALSE;
		ID5_SETUP :=FALSE;
	
		TMR1(IN:=FALSE);
		TMR2(IN:=FALSE);
		TMR3(IN:=FALSE);
		TMR4(IN:=FALSE);
		TMR5(IN:=FALSE);
	//ACTIVE_ID:=1;
	//FUKUDA_RUNNING:=TRUE;
		INPUT_VAR.FUKUDA_HOME:=TRUE;
	END_IF
	
	ELSE
				
	ID1_SVON :=TRUE;
	ID2_SVON :=TRUE;
	ID3_SVON :=TRUE;
	ID4_SVON :=TRUE;
	ID5_SVON :=TRUE;

	END_IF
ELSE
	TMR6(IN:=FALSE);

	CASE INPUT_VAR.ACTIVE_ID OF
	0:
		INPUT_VAR.I_CASE:=INPUT_VAR.I_CASE+1;
		//INPUT_VAR.I_FUKUDA_RUNNING:=FALSE;
		INPUT_VAR.ACTIVE_ID:=6;
		
	1:
		IF STEP_DATA_1 = 0 THEN
			INPUT_VAR.ACTIVE_ID:=2;
		ELSE
			IF ID1_ALARM THEN
				Reset := TRUE;
				TMR10(IN:=TRUE,PT:= PROCESS_DELAY);
				IF TMR10.Q THEN
					Reset := FALSE;
				END_IF
			ELSE
				ID1_StepData :=STEP_DATA_1;
				ID1_Drive := FALSE;
				TMR11(IN:=TRUE,PT:= PROCESS_DELAY);
				IF TMR11.Q THEN
					IF ID1_INP THEN
					ID1_Drive := TRUE;
					TMR12(IN:=TMR11.Q,PT:= PROCESS_DELAY);
					IF TMR12.Q THEN
						ID1_Drive := FALSE;
						INPUT_VAR.ACTIVE_ID:=2;
						TMR10(IN:=FALSE);
						TMR11(IN:=FALSE);
						TMR12(IN:=FALSE);
						INPUT_VAR.FUKUDA_HOME:=TRUE;
					END_IF
					ELSE
					INPUT_VAR.ACTIVE_ID:=1;
					END_IF
					
				END_IF
			END_IF
		END_IF
	//	INPUT_VAR.I_CASE:=INPUT_VAR.I_CASE+1;
		//INPUT_VAR.I_FUKUDA_RUNNING:=FALSE;
	2:
		IF STEP_DATA_2 = 0 THEN
			INPUT_VAR.ACTIVE_ID:=3;
		ELSE
			
			IF ID2_ALARM THEN
				Reset := TRUE;
				TMR20(IN:=TRUE,PT:= PROCESS_DELAY);
				IF TMR20.Q THEN
					Reset := FALSE;
				END_IF
			ELSE
			ID2_StepData :=STEP_DATA_2;
			TMR21(IN:=TRUE,PT:= PROCESS_DELAY);
			IF TMR21.Q THEN
				ID2_Drive := TRUE;
				TMR22(IN:=TMR21.Q,PT:= PROCESS_DELAY);
				IF TMR22.Q THEN
				IF ID2_INP THEN
					ID2_Drive := FALSE;
					INPUT_VAR.ACTIVE_ID:=3;
					TMR20(IN:=FALSE);
					TMR21(IN:=FALSE);
					TMR22(IN:=FALSE);
					ELSE
					INPUT_VAR.ACTIVE_ID:=2;
				END_IF
				END_IF
			END_IF
			END_IF
		END_IF
	3:
		IF STEP_DATA_3 = 0 THEN
			INPUT_VAR.ACTIVE_ID:=4;
		ELSE
			
		IF ID3_ALARM THEN
			Reset := TRUE;
			TMR30(IN:=START_PROCESS,PT:= PROCESS_DELAY);
			IF TMR30.Q THEN
				Reset := FALSE;
			END_IF
		ELSE
		
		ID3_StepData :=STEP_DATA_3;
		TMR31(IN:=TRUE,PT:= PROCESS_DELAY);
		IF TMR31.Q THEN
			ID3_DRIVE := TRUE;	
			TMR32(IN:=TMR31.Q,PT:= PROCESS_DELAY);
			
			IF TMR32.Q THEN
				IF  ID3_INP THEN
				ID3_Drive := FALSE;
				INPUT_VAR.ACTIVE_ID:=4;
				TMR30(IN:=FALSE);
				TMR31(IN:=FALSE);
				TMR32(IN:=FALSE);
				ELSE
					INPUT_VAR.ACTIVE_ID:=3;
				END_IF
			END_IF
		END_IF
		END_IF
	END_IF
4:
		IF STEP_DATA_4 = 0 THEN
			INPUT_VAR.ACTIVE_ID:=5;
		ELSE
			IF ID4_ALARM THEN
				Reset := TRUE;
				TMR40(IN:=TRUE,PT:= PROCESS_DELAY);
				IF TMR40.Q THEN
					Reset := FALSE;
				END_IF
			ELSE
				IF NOT ID4_READY THEN
					ID4_SETUP :=TRUE;
					IF ID4_INP THEN
						ID4_READY:=TRUE;
					END_IF
				ELSE
					ID4_StepData :=STEP_DATA_4;
					TMR41(IN:=TRUE,PT:= PROCESS_DELAY);
					IF TMR41.Q THEN
						ID4_Drive := TRUE;
						TMR42(IN:=TMR41.Q,PT:= PROCESS_DELAY);
						IF TMR42.Q THEN
							IF ID4_INP THEN
								ID4_Drive := FALSE;
								INPUT_VAR.ACTIVE_ID:=5;
								TMR40(IN:=FALSE);
								TMR41(IN:=FALSE);
								TMR42(IN:=FALSE);
							ELSE
								INPUT_VAR.ACTIVE_ID:=4;
							END_IF
						END_IF
					END_IF
				END_IF
			END_IF
		END_IF
	5:
		IF STEP_DATA_5 = 0 THEN
			INPUT_VAR.ACTIVE_ID:=0;
		ELSE
			
			IF ID5_ALARM THEN
				Reset := TRUE;
				TMR50(IN:=TRUE,PT:= PROCESS_DELAY);
				IF TMR50.Q THEN
					Reset := FALSE;
				END_IF
			ELSE
				IF NOT ID5_READY THEN
					ID5_SETUP :=TRUE;
					IF ID5_INP THEN
						ID5_READY:=TRUE;
					END_IF
				ELSE
					ID5_StepData :=STEP_DATA_5;
					TMR51(IN:=TRUE,PT:= PROCESS_DELAY);
					IF TMR51.Q THEN
						ID5_Drive := TRUE;	
						TMR52(IN:=TMR51.Q,PT:= PROCESS_DELAY);
						IF TMR52.Q THEN
							IF ID5_INP THEN
								ID5_Drive := FALSE;
								INPUT_VAR.ACTIVE_ID:=0;
								TMR50(IN:=FALSE);
								TMR51(IN:=FALSE);
								TMR52(IN:=FALSE);
							ELSE
								INPUT_VAR.ACTIVE_ID:=5;
							END_IF
						END_IF
					END_IF
				END_IF
			END_IF
		END_IF
END_CASE 

	//START_PROCESS := FALSE;
END_IF
TMR7(IN:=reset,PT:= T#1S);
IF  tmr7.Q THEN
	reset:=FALSE;
END_IF
IF ID1_ALARM OR ID2_ALARM OR ID3_ALARM OR ID4_ALARM OR ID5_ALARM THEN
	reset:=TRUE;
	INPUT_VAR.ALARM1:=ID1_ALARM OR ID2_ALARM OR ID3_ALARM OR ID4_ALARM OR ID5_ALARM;
ELSE
	reset:=FALSE;
END_IF
IF reset THEN
	ID1_Reset := TRUE;
	ID2_Reset := TRUE;
	ID3_Reset := TRUE;
	ID4_Reset := TRUE;
	ID5_Reset := TRUE;
	TMR_ACTIVATE_RESET(IN:=TRUE,PT:=T#10S);
	IF TMR_ACTIVATE_RESET.Q THEN
		TMR_RES_CARTSN(IN:=TRUE,PT:=T#0.5S);
	END_IF
	
ELSE
	TMR_ACTIVATE_RESET(IN:=FALSE);
	TMR_RES_CARTSN(IN:=FALSE);
	ID1_Reset := FALSE;
	ID2_Reset := FALSE;
	ID3_Reset := FALSE;
	ID4_Reset := FALSE;
	ID5_Reset := FALSE;
END_IF
INPUT_VAR.O_RESET_CARTESSIAN := TMR_RES_CARTSN.Q;

END_PROGRAM

// ---- POUs/FUKUDA/FUKUDA_MOVE_1.TcPOU
PROGRAM FUKUDA_MOVE_1
//FUNCTION FUKUDA_MOVE : BOOL
VAR_INPUT
	STEP_DATA_1: BYTE;
	STEP_DATA_2: BYTE;
	STEP_DATA_3: BYTE;
	STEP_DATA_4: BYTE;
	STEP_DATA_5: BYTE;
	FUKUDA_HOME: INT;
END_VAR

VAR
	
	(*
	DataWordInput1 AT %IB100 : ARRAY [0..15] OF WORD; 
	DataWordInput2 AT %IB132 : ARRAY [16..31] OF WORD; 
	DataWordInput3 AT %IB164 : ARRAY [32..47] OF WORD; 
	DataWordInput4 AT %IB196 : ARRAY [48..56] OF WORD; 
	DataWordOutput1 AT %QB100 : ARRAY [0..15] OF WORD; 
	DataWordOutput2 AT %QB132 : ARRAY [16..31] OF WORD; 
	DataWordOutput3 AT %QB164 : ARRAY [32..47] OF WORD; 
	DataWordOutput4 AT %QB196 : ARRAY [48..56] OF WORD; 
	*)
	Gateway_Q0_MODE_COMMAND_0 AT %QX100.0 : BOOL ;
	Gateway_Q0_MODE_COMMAND_1 AT %QX100.1 : BOOL ;
	Gateway_Q0_RESET AT %QX100.4 : BOOL;
	Gateway_Q0_RESTART AT %QX100.5 : BOOL;
	Gateway_Q0_STOP AT %QX100.7 : BOOL;
	Gateway_Q1_0 AT %QX101.0 : BOOL;
	Gateway_Q1_1 AT %QX101.1 : BOOL;
	Gateway_Q1_2 AT %QX101.2 : BOOL;
	Gateway_Q1_3 AT %QX101.3 : BOOL;
	Gateway_Q1_4 AT %QX101.4 : BOOL;
	Gateway_Gateway_Unit_2_Status AT %QB102 : BYTE;
	Gateway_Q3_0 AT %QX103.0 : BOOL;
	Gateway_Q3_1 AT %QX103.1 : BOOL;
	Gateway_Q3_2 AT %QX103.2 : BOOL;
	Gateway_Q3_3 AT %QX103.3 : BOOL;	
	

	ID1_StepData AT %QB114 : BYTE;
	ID1_Hold AT %QX115.0 : BOOL;
	ID1_SVON AT %QX115.1 : BOOL;
	ID1_Drive AT %QX115.2 : BOOL;
	ID1_Reset AT %QX115.3 : BOOL;
	ID1_Setup AT %QX115.4 : BOOL;
	

	ID2_StepData AT %QB134 : BYTE;
	ID2_Hold AT %QX135.0 : BOOL;
	ID2_SVON AT %QX135.1 : BOOL;
	ID2_Drive AT %QX135.2 : BOOL;
	ID2_Reset AT %QX135.3 : BOOL;
	ID2_Setup AT %QX135.4 : BOOL;


	ID3_StepData AT %QB154 : BYTE;
	ID3_Hold AT %QX155.0 : BOOL;
	ID3_SVON AT %QX155.1 : BOOL;
	ID3_Drive AT %QX155.2 : BOOL;
	ID3_Reset AT %QX155.3 : BOOL;
	ID3_Setup AT %QX155.4 : BOOL;
	
	
	ID4_StepData AT %QB174 : BYTE;
	ID4_Hold AT %QX175.0 : BOOL;
	ID4_SVON AT %QX175.1 : BOOL;
	ID4_Drive AT %QX175.2 : BOOL;
	ID4_Reset AT %QX175.3 : BOOL;
	ID4_Setup AT %QX175.4 : BOOL;
	

	ID5_StepData AT %QB194 : BYTE;
	ID5_Hold AT %QX195.0 : BOOL;
	ID5_SVON AT %QX195.1 : BOOL;
	ID5_Drive AT %QX195.2 : BOOL;
	ID5_Reset AT %QX195.3 : BOOL;
	ID5_Setup AT %QX195.4 : BOOL;
	
	byte0 : BYTE;
	byte1 : BYTE;
	byte2 : BYTE;
	byte3 : BYTE;
	
	bit14_0 : BOOL;
	bit14_1 : BOOL;
	bit14_2 : BOOL;
	bit14_3 : BOOL;
	bit14_4 : BOOL;
	bit14_5 : BOOL;
	
	bit15_0 : BOOL;
	bit15_1 : BOOL;
	bit15_2 : BOOL;
	bit15_3 : BOOL;
	bit15_4 : BOOL; 
	
	bit34_0 : BOOL;
	bit34_1 : BOOL;
	bit34_2 : BOOL;
	bit34_3 : BOOL;
	bit34_4 : BOOL;
	bit34_5 : BOOL;
	
	bit35_0 : BOOL;
	bit35_1 : BOOL;
	bit35_2 : BOOL;
	bit35_3 : BOOL;
	bit35_4 : BOOL; 
	
	bit54_0 : BOOL;
	bit54_1 : BOOL;
	bit54_2 : BOOL;
	bit54_3 : BOOL;
	bit54_4 : BOOL;
	bit54_5 : BOOL;
	
	bit55_0 : BOOL;
	bit55_1 : BOOL;
	bit55_2 : BOOL;
	bit55_3 : BOOL;
	bit55_4 : BOOL; 
	
	bit74_0 : BOOL;
	bit74_1 : BOOL;
	bit74_2 : BOOL;
	bit74_3 : BOOL;
	bit74_4 : BOOL;
	bit74_5 : BOOL;
	
	bit75_0 : BOOL;
	bit75_1 : BOOL;
	bit75_2 : BOOL;
	bit75_3 : BOOL;
	bit75_4 : BOOL; 
	
	bit94_0 : BOOL;
	bit94_1 : BOOL;
	bit94_2 : BOOL;
	bit94_3 : BOOL;
	bit94_4 : BOOL;
	bit94_5 : BOOL;
	
	bit95_0 : BOOL;
	bit95_1 : BOOL;
	bit95_2 : BOOL;
	bit95_3 : BOOL;
	bit95_4 : BOOL; 	
	
	ID1_I0_MODE_COMMAND_0 AT %IX100.0 : BOOL :=0;
	ID1_I0_MODE_COMMAND_1 AT %IX100.1 : BOOL:=0;
	ID1_I0_READY AT %IX100.4 : BOOL;
	ID1_I0_ALARM AT %IX100.5 : BOOL;
	ID1_I0_INITIAL AT %IX100.6 : BOOL;
	ID1_I0_COMMUNICATING AT %IX100.7 : BOOL;
	ID1_I1_0 AT %IX101.0 : BOOL;
	ID1_I1_1 AT %IX101.1 : BOOL;
	ID1_I1_2 AT %IX101.2 : BOOL;
	ID1_I1_3 AT %IX101.3 : BOOL;
	ID1_I1_4 AT %IX101.4 : BOOL;
	ID1_I2_0 AT %IX102.0 : BOOL;
	ID1_I2_1 AT %IX102.1 : BOOL;
	ID1_I2_2 AT %IX102.2 : BOOL;
	ID1_I2_3 AT %IX102.3 : BOOL;
	ID1_I2_4 AT %IX102.4 : BOOL;

	ID1_I3_0 AT %IX103.0 : BOOL;
	ID1_I3_1 AT %IX103.1 : BOOL;
	
	ID1_I32_0 AT %IX132.0 : BOOL;
	ID1_I32_1 AT %IX132.1 : BOOL;
	ID1_I33_0 AT %IX133.0 : BOOL;
	ID1_I33_1 AT %IX133.1 : BOOL;
(*-----------------------------------------------------------*)

	iTest15: SINT;
	iTest16: SINT;
	
	bTest1 : BOOL;
	bTest2 : BOOL;
	bTest3 : BOOL;
	bTest4 : BOOL;
	bTest5 : BOOL;
	bTest6 : BOOL;
	bTest7 : BOOL;
	bTest8 : BOOL;
	bTest9 : BOOL;
	bTest10 : BOOL;
	bTest11 : BOOL;
	bTest12 : BOOL;
	bTest13 : BOOL;
	bTest14 : BOOL;
	
	StepData1 : BYTE;
	StepData2 : BYTE;
	StepData3 : BYTE;
	StepData4 : BYTE;
	StepData5 : BYTE;
	
	star :BOOL;
	hom : BOOL;

	reset: BOOL;
	
	ID1_ALARM AT%IX115.7 : BOOL;
	ID2_ALARM AT%IX135.7 : BOOL;
	ID3_ALARM AT%IX155.7 : BOOL;
	ID4_ALARM AT%IX175.7 : BOOL;
	ID5_ALARM AT%IX195.7 : BOOL;
	
	ID1_SVRE AT%IX115.1 : BOOL;
	ID2_SVRE AT%IX135.1 : BOOL;
	ID3_SVRE AT%IX155.1 : BOOL;
	ID4_SVRE AT%IX175.1 : BOOL;
	ID5_SVRE AT%IX195.1 : BOOL;
	
	ID1_INP AT%IX115.3 : BOOL;
	ID2_INP AT%IX135.3 : BOOL;
	ID3_INP AT%IX155.3 : BOOL;
	ID4_INP AT%IX175.3 : BOOL;
	ID5_INP AT%IX195.3 : BOOL;
	
	PROSES: STRING;
	STAGE: INT;
	
	PROCESS: INT;
	START_PROCESS: BOOL;
	STEP_DATAS: INT;
	PROCESS_DELAY: TIME :=T#300MS;
	FUKUDA_RUNNING: BOOL :=FALSE;
	ACTIVE_STEPDATA : BYTE;
	//ACTIVE_ID: INT :=1;
	TMR1: TON;
	TMR2: TON;
	TMR3: TON;
	TMR4: TON;
	TMR5: TON;
	TMR6: TON;
	TMR10: Ton;
	TMR11: TON;
	TMR12: TON;
	TMR13: TON;
	TMR14: TON;
	TMR20: TON;
	TMR21: TON;
	TMR22: TON;
	TMR23: TON;
	TMR30: TON;
	TMR31: TON;
	TMR32: TON;
	TMR33: TON;
	TMR40: TON;
	TMR41: TON;
	TMR42: TON;
	TMR43: TON;
	TMR50: TON;
	TMR51: TON;
	TMR52: TON;
	TMR53: TON;
	
	
	TMR101: TON;
	TMR102: TON;
	TMR103: TON;
	TMR104: TON;
	TMR105: TON;
	TMR106: TON;
	ID5: INT;
	TMR7: Ton;
	TMR_RES_CARTSN: TOF;
	TMR_ACTIVATE_RESET: TON;
END_VAR


PROCESS_DELAY:= T#400MS;
IF 	INPUT_VAR.ACTIVE_ID >=0 THEN
STEP_DATA_1:=STEP_DATA_1+1;

IF STEP_DATA_2>=5 THEN
	STEP_DATA_2:=STEP_DATA_2+1;
END_IF

STEP_DATA_3:=STEP_DATA_3+1;	
END_IF


IF NOT INPUT_VAR.FUKUDA_HOME THEN //fukuda_running THEN
	IF  ID1_SVRE AND ID2_SVRE  AND  ID3_SVRE AND  ID4_SVRE AND  ID5_SVRE THEN
		TMR1(IN:=TRUE,PT:=T#0.5S);
		TMR4(IN:=TRUE,PT:=T#3S);
		TMR5(IN:=TRUE,PT:=T#3.5S);
		TMR6(IN:=TRUE,PT:=T#25S);
		IF ID1_SVRE THEN
			ID1_SETUP :=TMR5.Q;
		ELSE
			ID1_SVON :=TRUE;	
		END_IF

		IF ID2_SVRE THEN
			ID2_SETUP :=TMR1.Q;
		ELSE
			ID2_SVON :=TRUE;	
		END_IF
	
		IF ID3_SVRE THEN
		ID3_SETUP :=TMR4.Q;
		ELSE
			ID3_SVON :=TRUE;	
		END_IF
		CASE INPUT_VAR.I_CURRENT_TRANSACTION.TRANSPORT_INDEX OF
		1:
			TMR2(IN:=TRUE,PT:=T#1S);
			IF ID4_SVRE THEN
				ID4_SETUP :=TMR2.Q;
			ELSE
				ID4_SVON :=TRUE;	
			END_IF
		2:
			TMR3(IN:=TRUE,PT:=T#1.5S);
			IF ID5_SVRE THEN
				ID5_SETUP :=TMR3.Q;
			ELSE
				ID5_SVON :=TRUE;	
			END_IF
		END_CASE

	//IF TMR6.Q THEN
	IF ID1_INP AND ID2_INP AND ID3_INP AND (ID4_INP OR ID5_INP) THEN
		ID1_SETUP :=FALSE;
		ID2_SETUP :=FALSE;
		ID3_SETUP :=FALSE;
		ID4_SETUP :=FALSE;
		ID5_SETUP :=FALSE;
	
		TMR1(IN:=FALSE);
		TMR2(IN:=FALSE);
		TMR3(IN:=FALSE);
		TMR4(IN:=FALSE);
		TMR5(IN:=FALSE);
	//ACTIVE_ID:=1;
	//FUKUDA_RUNNING:=TRUE;
		INPUT_VAR.FUKUDA_HOME:=TRUE;
	END_IF
	
	ELSE
				
	ID1_SVON :=TRUE;
	ID2_SVON :=TRUE;
	ID3_SVON :=TRUE;
	ID4_SVON :=TRUE;
	ID5_SVON :=TRUE;

	END_IF
ELSE
	TMR6(IN:=FALSE);

	CASE INPUT_VAR.ACTIVE_ID OF
	0:
		INPUT_VAR.I_CASE:=INPUT_VAR.I_CASE+1;
		//INPUT_VAR.I_FUKUDA_RUNNING:=FALSE;
		INPUT_VAR.ACTIVE_ID:=6;
		
	1:
		IF STEP_DATA_1 = 0 THEN
			INPUT_VAR.ACTIVE_ID:=2;
		ELSE
			IF ID1_ALARM THEN
				Reset := TRUE;
				TMR10(IN:=TRUE,PT:= PROCESS_DELAY);
				IF TMR10.Q THEN
					Reset := FALSE;
				END_IF
			ELSE
				ID1_StepData :=STEP_DATA_1;
				ID1_Drive := FALSE;
				TMR11(IN:=TRUE,PT:= PROCESS_DELAY);
				IF TMR11.Q THEN
					IF ID1_INP THEN
					ID1_Drive := TRUE;
					TMR12(IN:=TMR11.Q,PT:= PROCESS_DELAY);
					IF TMR12.Q THEN
						ID1_Drive := FALSE;
						INPUT_VAR.ACTIVE_ID:=2;
						TMR10(IN:=FALSE);
						TMR11(IN:=FALSE);
						TMR12(IN:=FALSE);
						INPUT_VAR.FUKUDA_HOME:=TRUE;
					END_IF
					ELSE
					INPUT_VAR.ACTIVE_ID:=1;
					END_IF
					
				END_IF
			END_IF
		END_IF
	//	INPUT_VAR.I_CASE:=INPUT_VAR.I_CASE+1;
		//INPUT_VAR.I_FUKUDA_RUNNING:=FALSE;
	2:
		IF STEP_DATA_2 = 0 THEN
			INPUT_VAR.ACTIVE_ID:=3;
		ELSE
			
			IF ID2_ALARM THEN
				Reset := TRUE;
				TMR20(IN:=TRUE,PT:= PROCESS_DELAY);
				IF TMR20.Q THEN
					Reset := FALSE;
				END_IF
			ELSE
			ID2_StepData :=STEP_DATA_2;
			TMR21(IN:=TRUE,PT:= PROCESS_DELAY);
			IF TMR21.Q THEN
				ID2_Drive := TRUE;
				TMR22(IN:=TMR21.Q,PT:= PROCESS_DELAY);
				IF TMR22.Q THEN
				IF ID2_INP THEN
					ID2_Drive := FALSE;
					INPUT_VAR.ACTIVE_ID:=3;
					TMR20(IN:=FALSE);
					TMR21(IN:=FALSE);
					TMR22(IN:=FALSE);
					ELSE
					INPUT_VAR.ACTIVE_ID:=2;
				END_IF
				END_IF
			END_IF
			END_IF
		END_IF
	3:
		IF STEP_DATA_3 = 0 THEN
			INPUT_VAR.ACTIVE_ID:=4;
		ELSE
			
		IF ID3_ALARM THEN
			Reset := TRUE;
			TMR30(IN:=START_PROCESS,PT:= PROCESS_DELAY);
			IF TMR30.Q THEN
				Reset := FALSE;
			END_IF
		ELSE
		
		ID3_StepData :=STEP_DATA_3;
		TMR31(IN:=TRUE,PT:= PROCESS_DELAY);
		IF TMR31.Q THEN
			ID3_DRIVE := TRUE;	
			TMR32(IN:=TMR31.Q,PT:= PROCESS_DELAY);
			
			IF TMR32.Q THEN
				IF  ID3_INP THEN
				ID3_Drive := FALSE;
				INPUT_VAR.ACTIVE_ID:=4;
				TMR30(IN:=FALSE);
				TMR31(IN:=FALSE);
				TMR32(IN:=FALSE);
				ELSE
					INPUT_VAR.ACTIVE_ID:=3;
				END_IF
			END_IF
		END_IF
		END_IF
	END_IF
4:
		IF STEP_DATA_4 = 0 THEN
			INPUT_VAR.ACTIVE_ID:=5;
		ELSE
			IF ID4_ALARM THEN
				Reset := TRUE;
				TMR40(IN:=TRUE,PT:= PROCESS_DELAY);
				IF TMR40.Q THEN
					Reset := FALSE;
				END_IF
			ELSE
			
			ID4_StepData :=STEP_DATA_4;
			TMR41(IN:=TRUE,PT:= PROCESS_DELAY);
			IF TMR41.Q THEN
				ID4_Drive := TRUE;
				TMR42(IN:=TMR41.Q,PT:= PROCESS_DELAY);
				
				IF TMR42.Q THEN
					IF ID4_INP THEN
					ID4_Drive := FALSE;
					INPUT_VAR.ACTIVE_ID:=5;
					TMR40(IN:=FALSE);
					TMR41(IN:=FALSE);
					TMR42(IN:=FALSE);
					ELSE
						INPUT_VAR.ACTIVE_ID:=4;
					END_IF
				END_IF
			END_IF
			END_IF
		END_IF
	5:
		IF STEP_DATA_5 = 0 THEN
			INPUT_VAR.ACTIVE_ID:=0;
		ELSE
			
			IF ID5_ALARM THEN
				Reset := TRUE;
				TMR50(IN:=TRUE,PT:= PROCESS_DELAY);
				IF TMR50.Q THEN
					Reset := FALSE;
				END_IF
			ELSE
			
			ID5_StepData :=STEP_DATA_5;
			TMR51(IN:=TRUE,PT:= PROCESS_DELAY);
			IF TMR51.Q THEN
				ID5_Drive := TRUE;	
				TMR52(IN:=TMR51.Q,PT:= PROCESS_DELAY);
				IF TMR52.Q THEN
					IF ID5_INP THEN
					ID5_Drive := FALSE;
					INPUT_VAR.ACTIVE_ID:=0;
					TMR50(IN:=FALSE);
					TMR51(IN:=FALSE);
					TMR52(IN:=FALSE);
					ELSE
					INPUT_VAR.ACTIVE_ID:=5;
				END_IF
			END_IF
			END_IF
		END_IF
		END_IF
END_CASE 

	//START_PROCESS := FALSE;
END_IF
TMR7(IN:=reset,PT:= T#1S);
IF  tmr7.Q THEN
	reset:=FALSE;
END_IF
IF ID1_ALARM OR ID2_ALARM OR ID3_ALARM OR ID4_ALARM OR ID5_ALARM THEN
			reset:=TRUE;
			ELSE
				reset:=FALSE;
			END_IF
IF reset THEN
	ID1_Reset := TRUE;
	ID2_Reset := TRUE;
	ID3_Reset := TRUE;
	ID4_Reset := TRUE;
	ID5_Reset := TRUE;
	TMR_ACTIVATE_RESET(IN:=TRUE,PT:=T#10S);
	IF TMR_ACTIVATE_RESET.Q THEN
		TMR_RES_CARTSN(IN:=TRUE,PT:=T#0.5S);
	END_IF
	
ELSE
	TMR_ACTIVATE_RESET(IN:=FALSE);
	TMR_RES_CARTSN(IN:=FALSE);
	ID1_Reset := FALSE;
	ID2_Reset := FALSE;
	ID3_Reset := FALSE;
	ID4_Reset := FALSE;
	ID5_Reset := FALSE;
END_IF
INPUT_VAR.O_RESET_CARTESSIAN := TMR_RES_CARTSN.Q;

END_PROGRAM

// ---- POUs/FUKUDA/INPUT_PROG.TcPOU
PROGRAM INPUT_PROG
VAR
	T1: TON;
	
	T2: TON;
	Q: BOOL;
	OUT1: BOOL;
	AR: R_TRIG;
	LOTBOX_STAT: BOOL;
	RTRIG_1: F_TRIG;
	RTRIG_2: F_TRIG;
	RTRIG_3: F_TRIG;
	RTRIG_4: F_TRIG;
	QUEUE_INDEX_1: INT;
	QUEUE_INDEX_2: INT;
	QUEUE_INDEX_3: INT;
	QUEUE_INDEX_4: INT;
	IC_CASE: INT;
	TMR1: TON;
	TMR2: TON;
	I_STOPPER_TRANSFER_A: INT;
	TMR3: TON;
	TMR4: TON;
	TMR5: TON;
	TMR6: TON;
	TMR7: TON;
	TMR8: TON;
	TMR9: TON;
	TMR10: TON;
	TMR11: TON;
	TMR12: TON;
	TMR14: TON;
	COUNTER_1: CTU;
	RESET_COUNTER: BOOL;
	COUNTER_2: CTU;
	PULS1: TON;
	PULSE_OUT1: TON;
	TP1: TON;
	PULSE_OUT2: TON;
	PULS2: TON;
	PULS3: TON;
	CNTFUKUDA: BYTE;
	CNTFUKUDAB: BYTE;
	CNTFUKUDAA: BYTE;
	LOTBOX_TEMPI1: INT;
	LOTBOX_TEMPI2: INT;
	LOTBOX_TEMPI3: INT;
	LOTBOX_TEMPI4: INT;
	LOTBOX_ACCI: INT;
END_VAR

VAR PERSISTENT
	AR_TRIG: R_TRIG;
END_VAR


IF CNTFUKUDAA >=20 THEN
	//INPUT_VAR.I_FUKUDA_TRANSFER_A_PICK_DONE:=TRUE;
	CNTFUKUDAA:=0;
	ELSE
	CNTFUKUDAA:=INPUT_G6_VAR.COUNTER_FUKUDA_A;
END_IF

IF CNTFUKUDAB >=20 THEN
	//INPUT_VAR.I_FUKUDA_TRANSFER_B_PICK_DONE:=TRUE;
	CNTFUKUDAB:=0;
	ELSE
	CNTFUKUDAB:=INPUT_G6_VAR.COUNTER_FUKUDA_B;
END_IF


IF NOT INPUT_VAR.I_LOTBOX_DETECT_1 OR NOT INPUT_VAR.I_LOTBOX_DETECT_2 OR NOT INPUT_VAR.I_LOTBOX_DETECT_3 OR NOT INPUT_VAR.I_LOTBOX_DETECT_4 THEN
	INPUT_VAR.O_TOWER_LAMP_YELLOW :=TRUE;
END_IF 


IF FLAG_VAR.ALLOW_EXECUTE_LOAD_FUKUDA THEN 
	IF INPUT_VAR.I_CASE=100 OR INPUT_VAR.I_CASE=12 THEN
		INPUT_VAR.I_CASE:=0;
		IC_CASE:=0;	
		END_IF			
	LOAD_FUKUDA();
END_IF
IF FLAG_VAR.ALLOW_EXECUTE_RETURN_FUKUDA THEN 
	IF INPUT_VAR.I_CASE=100 THEN
		INPUT_VAR.I_CASE:=0;
		IC_CASE:=0;
	END_IF	
	RETURN_FUKUDA();	
END_IF

(*
TMR4(IN:=INPUT_VAR.I_FUKUDA_TRANSFER_AT_FRONT_B,PT:= T#2S);
TMR5(IN:=INPUT_VAR.I_STOPPER_TRANSFER_ON_B,PT:=T#2S);
TMR6(IN:=INPUT_G6_VAR.O_G6_SELECT_FUKUDA_B,PT:=T#10S);

INPUT_VAR.O_STOPPER_TRANSFER_B:=TMR4.Q;
INPUT_G6_VAR.O_G6_SELECT_FUKUDA_B:=TMR5.Q;
*)

//END_IF
//LOTBOX_STAT := INPUT_VAR.I_LOTBOX_DETECT_1 + INPUT_VAR.I_LOTBOX_DETECT_2 + INPUT_VAR.I_LOTBOX_DETECT_3 + INPUT_VAR.I_LOTBOX_DETECT_4 


//INPUT_G6_VAR.I_G6_HOME:=POWER_CONTROL.O_PWR_CTRL_ROBOT_G6;
//INDEXING1_VAR.I_INDEXING_HOME := POWER_CONTROL.O_PWR_CTRL_INDEXING_1;

